Yaskawa INFORM job: A_ROOF_UPPER_0614_2_PAINT_30.JBI

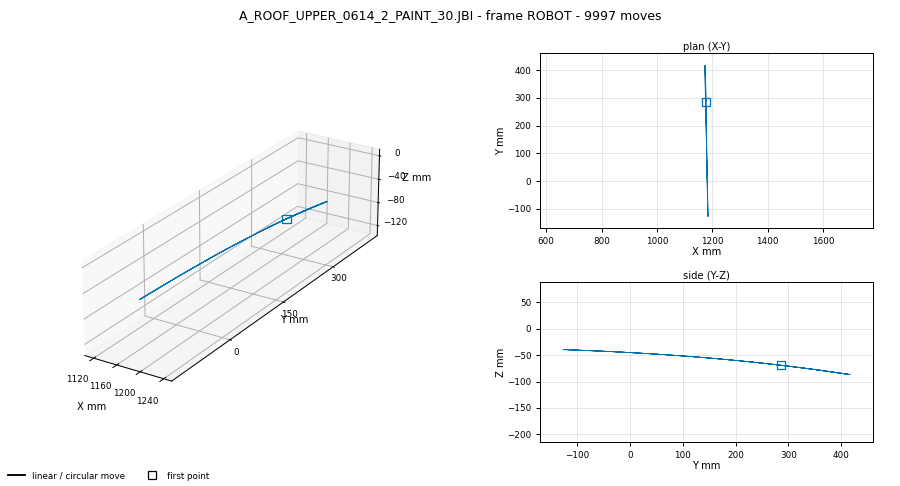
[picture p0: tool path of A_ROOF_UPPER_0614_2_PAINT_30.JBI in frame ROBOT, 9997 of 9997 moves have a stored position in this frame; points joined in program order, loops and branches not executed]
/JOB
//NAME A_ROOF_UPPER_0614_2_PAINT30
//POS
///NPOS 9997,0,0,0,0,0
///TOOL 1
///USER 0
///POSTYPE ROBOT
///RECTAN
///RCONF 1,0,0,0,0,0,0,0,0,0,0,0,0,0,0,0,0,0,0,0,0,0,0,0
C00000=1177.111,285.964,-68.993,-176.930,7.670,148.574
C00001=1177.106,286.213,-69.022,-176.928,7.672,148.574
C00002=1177.102,286.461,-69.051,-176.925,7.675,148.574
C00003=1177.098,286.710,-69.081,-176.922,7.678,148.574
C00004=1177.093,286.957,-69.110,-176.920,7.681,148.574
C00005=1177.089,287.205,-69.139,-176.917,7.684,148.574
C00006=1177.085,287.454,-69.169,-176.914,7.687,148.574
C00007=1177.081,287.702,-69.198,-176.912,7.690,148.574
C00008=1177.076,287.977,-69.230,-176.909,7.694,148.574
C00009=1177.071,288.251,-69.263,-176.906,7.697,148.574
C00010=1177.067,288.526,-69.295,-176.904,7.700,148.574
C00011=1177.062,288.801,-69.329,-176.901,7.703,148.574
C00012=1177.058,289.049,-69.358,-176.898,7.705,148.574
C00013=1177.053,289.297,-69.387,-176.896,7.708,148.574
C00014=1177.049,289.545,-69.417,-176.893,7.711,148.574
C00015=1177.045,289.793,-69.446,-176.890,7.714,148.574
C00016=1177.040,290.042,-69.476,-176.887,7.717,148.574
C00017=1177.036,290.290,-69.506,-176.885,7.720,148.574
C00018=1177.032,290.538,-69.535,-176.883,7.723,148.574
C00019=1177.027,290.787,-69.565,-176.880,7.726,148.574
C00020=1177.023,291.035,-69.594,-176.877,7.729,148.574
C00021=1177.019,291.283,-69.623,-176.875,7.732,148.574
C00022=1177.015,291.531,-69.653,-176.872,7.735,148.574
C00023=1177.011,291.780,-69.682,-176.869,7.738,148.574
C00024=1177.006,292.028,-69.713,-176.867,7.741,148.574
C00025=1177.002,292.276,-69.743,-176.865,7.743,148.574
C00026=1176.998,292.524,-69.772,-176.862,7.746,148.574
C00027=1176.994,292.772,-69.801,-176.859,7.749,148.574
C00028=1176.989,293.021,-69.831,-176.857,7.752,148.574
C00029=1176.985,293.269,-69.862,-176.854,7.755,148.574
C00030=1176.981,293.517,-69.891,-176.852,7.759,148.574
C00031=1176.976,293.765,-69.921,-176.849,7.761,148.574
C00032=1176.972,294.014,-69.950,-176.847,7.764,148.574
C00033=1176.968,294.261,-69.980,-176.844,7.767,148.574
C00034=1176.963,294.510,-70.010,-176.841,7.770,148.574
C00035=1176.959,294.758,-70.040,-176.839,7.773,148.574
C00036=1176.955,295.006,-70.070,-176.836,7.776,148.574
C00037=1176.950,295.254,-70.100,-176.834,7.779,148.574
C00038=1176.946,295.503,-70.129,-176.831,7.782,148.574
C00039=1176.942,295.750,-70.160,-176.828,7.785,148.574
C00040=1176.938,295.998,-70.189,-176.826,7.787,148.574
C00041=1176.933,296.247,-70.219,-176.824,7.790,148.574
C00042=1176.929,296.495,-70.249,-176.821,7.793,148.574
C00043=1176.925,296.743,-70.279,-176.818,7.796,148.574
C00044=1176.921,296.991,-70.309,-176.815,7.799,148.574
C00045=1176.916,297.239,-70.339,-176.813,7.802,148.574
C00046=1176.913,297.488,-70.369,-176.810,7.806,148.574
C00047=1176.908,297.736,-70.399,-176.808,7.809,148.574
C00048=1176.904,297.984,-70.429,-176.805,7.812,148.574
C00049=1176.900,298.232,-70.459,-176.803,7.814,148.574
C00050=1176.895,298.481,-70.489,-176.801,7.817,148.574
C00051=1176.891,298.728,-70.519,-176.798,7.820,148.574
C00052=1176.886,298.977,-70.549,-176.795,7.823,148.574
C00053=1176.883,299.224,-70.580,-176.792,7.826,148.574
C00054=1176.878,299.473,-70.609,-176.790,7.829,148.574
C00055=1176.874,299.721,-70.640,-176.787,7.832,148.574
C00056=1176.871,299.969,-70.670,-176.785,7.835,148.574
C00057=1176.866,300.218,-70.700,-176.782,7.838,148.574
C00058=1176.862,300.465,-70.731,-176.780,7.842,148.574
C00059=1176.857,300.714,-70.761,-176.777,7.844,148.574
C00060=1176.853,300.961,-70.791,-176.775,7.847,148.574
C00061=1176.848,301.209,-70.821,-176.772,7.850,148.574
C00062=1176.844,301.458,-70.851,-176.770,7.853,148.574
C00063=1176.840,301.706,-70.882,-176.767,7.856,148.574
C00064=1176.836,301.954,-70.912,-176.764,7.859,148.574
C00065=1176.831,302.203,-70.942,-176.762,7.862,148.574
C00066=1176.827,302.450,-70.972,-176.759,7.865,148.574
C00067=1176.823,302.698,-71.003,-176.757,7.868,148.574
C00068=1176.819,302.947,-71.033,-176.754,7.871,148.574
C00069=1176.815,303.195,-71.064,-176.751,7.874,148.574
C00070=1176.811,303.443,-71.094,-176.749,7.877,148.574
C00071=1176.806,303.691,-71.125,-176.747,7.880,148.574
C00072=1176.802,303.939,-71.155,-176.744,7.883,148.574
C00073=1176.798,304.188,-71.185,-176.742,7.886,148.575
C00074=1176.793,304.436,-71.216,-176.739,7.889,148.575
C00075=1176.789,304.683,-71.246,-176.736,7.892,148.575
C00076=1176.785,304.931,-71.277,-176.733,7.895,148.574
C00077=1176.780,305.179,-71.308,-176.731,7.898,148.575
C00078=1176.777,305.427,-71.338,-176.728,7.901,148.575
C00079=1176.772,305.676,-71.368,-176.726,7.904,148.575
C00080=1176.767,305.924,-71.399,-176.723,7.907,148.575
C00081=1176.764,306.172,-71.429,-176.721,7.910,148.575
C00082=1176.760,306.420,-71.460,-176.718,7.913,148.575
C00083=1176.755,306.668,-71.491,-176.716,7.916,148.575
C00084=1176.751,306.916,-71.521,-176.714,7.919,148.575
C00085=1176.746,307.164,-71.552,-176.711,7.922,148.575
C00086=1176.742,307.413,-71.583,-176.709,7.925,148.575
C00087=1176.739,307.660,-71.613,-176.706,7.928,148.575
C00088=1176.734,307.908,-71.644,-176.703,7.931,148.575
C00089=1176.730,308.157,-71.675,-176.701,7.935,148.575
C00090=1176.725,308.405,-71.706,-176.698,7.937,148.575
C00091=1176.721,308.652,-71.736,-176.695,7.940,148.575
C00092=1176.717,308.901,-71.767,-176.693,7.944,148.575
C00093=1176.713,309.149,-71.798,-176.690,7.947,148.575
C00094=1176.708,309.397,-71.829,-176.688,7.950,148.575
C00095=1176.704,309.645,-71.859,-176.685,7.953,148.576
C00096=1176.700,309.893,-71.890,-176.683,7.956,148.576
C00097=1176.696,310.141,-71.921,-176.680,7.959,148.576
C00098=1176.691,310.389,-71.952,-176.678,7.962,148.576
C00099=1176.688,310.637,-71.983,-176.675,7.965,148.576
C00100=1176.684,310.885,-72.014,-176.672,7.968,148.576
C00101=1176.680,311.134,-72.045,-176.671,7.971,148.576
C00102=1176.675,311.382,-72.076,-176.668,7.974,148.576
C00103=1176.670,311.629,-72.106,-176.665,7.977,148.576
C00104=1176.667,311.878,-72.138,-176.663,7.980,148.576
C00105=1176.663,312.125,-72.168,-176.660,7.983,148.576
C00106=1176.658,312.373,-72.199,-176.658,7.986,148.576
C00107=1176.654,312.622,-72.230,-176.655,7.989,148.576
C00108=1176.650,312.869,-72.262,-176.652,7.992,148.576
C00109=1176.646,313.118,-72.293,-176.650,7.996,148.576
C00110=1176.641,313.366,-72.324,-176.647,7.999,148.576
C00111=1176.637,313.613,-72.355,-176.645,8.002,148.577
C00112=1176.632,313.890,-72.389,-176.642,8.006,148.577
C00113=1176.627,314.167,-72.424,-176.639,8.009,148.577
C00114=1176.623,314.444,-72.459,-176.637,8.012,148.577
C00115=1176.618,314.721,-72.493,-176.634,8.016,148.577
C00116=1176.614,314.969,-72.525,-176.631,8.019,148.577
C00117=1176.610,315.217,-72.556,-176.629,8.022,148.577
C00118=1176.605,315.464,-72.588,-176.626,8.025,148.577
C00119=1176.601,315.713,-72.619,-176.624,8.028,148.577
C00120=1176.597,315.961,-72.649,-176.621,8.031,148.577
C00121=1176.593,316.209,-72.681,-176.619,8.035,148.577
C00122=1176.588,316.457,-72.712,-176.616,8.038,148.577
C00123=1176.585,316.705,-72.744,-176.613,8.041,148.577
C00124=1176.580,316.953,-72.775,-176.611,8.044,148.578
C00125=1176.576,317.201,-72.807,-176.608,8.047,148.577
C00126=1176.572,317.449,-72.837,-176.606,8.050,148.578
C00127=1176.568,317.697,-72.869,-176.603,8.053,148.578
C00128=1176.564,317.945,-72.900,-176.601,8.057,148.578
C00129=1176.560,318.193,-72.932,-176.598,8.060,148.578
C00130=1176.555,318.441,-72.963,-176.596,8.063,148.578
C00131=1176.551,318.689,-72.994,-176.593,8.066,148.578
C00132=1176.547,318.936,-73.026,-176.590,8.069,148.578
C00133=1176.543,319.185,-73.057,-176.588,8.072,148.578
C00134=1176.539,319.432,-73.088,-176.585,8.075,148.578
C00135=1176.535,319.681,-73.120,-176.583,8.079,148.578
C00136=1176.531,319.929,-73.151,-176.581,8.081,148.578
C00137=1176.526,320.177,-73.184,-176.579,8.084,148.579
C00138=1176.522,320.425,-73.215,-176.576,8.087,148.579
C00139=1176.518,320.673,-73.246,-176.574,8.090,148.579
C00140=1176.514,320.921,-73.278,-176.571,8.093,148.579
C00141=1176.510,321.168,-73.309,-176.569,8.097,148.579
C00142=1176.506,321.417,-73.341,-176.566,8.100,148.579
C00143=1176.501,321.664,-73.372,-176.564,8.103,148.579
C00144=1176.497,321.912,-73.404,-176.560,8.107,148.579
C00145=1176.493,322.160,-73.436,-176.558,8.110,148.579
C00146=1176.489,322.408,-73.467,-176.555,8.113,148.579
C00147=1176.485,322.656,-73.499,-176.553,8.116,148.580
C00148=1176.481,322.904,-73.530,-176.550,8.119,148.580
C00149=1176.476,323.152,-73.563,-176.548,8.123,148.580
C00150=1176.473,323.400,-73.595,-176.546,8.126,148.580
C00151=1176.468,323.648,-73.625,-176.543,8.129,148.580
C00152=1176.464,323.896,-73.657,-176.541,8.132,148.580
C00153=1176.460,324.144,-73.690,-176.538,8.135,148.580
C00154=1176.455,324.392,-73.721,-176.536,8.139,148.580
C00155=1176.452,324.640,-73.753,-176.533,8.142,148.580
C00156=1176.448,324.888,-73.785,-176.531,8.145,148.581
C00157=1176.443,325.136,-73.817,-176.528,8.148,148.581
C00158=1176.439,325.384,-73.849,-176.526,8.151,148.581
C00159=1176.436,325.632,-73.881,-176.524,8.154,148.581
C00160=1176.431,325.879,-73.913,-176.521,8.157,148.581
C00161=1176.427,326.127,-73.945,-176.519,8.161,148.581
C00162=1176.423,326.375,-73.976,-176.516,8.164,148.581
C00163=1176.418,326.623,-74.009,-176.514,8.167,148.581
C00164=1176.414,326.871,-74.040,-176.511,8.170,148.581
C00165=1176.411,327.119,-74.072,-176.509,8.173,148.582
C00166=1176.406,327.367,-74.104,-176.506,8.177,148.582
C00167=1176.402,327.615,-74.136,-176.504,8.180,148.582
C00168=1176.398,327.863,-74.168,-176.501,8.183,148.582
C00169=1176.393,328.110,-74.200,-176.499,8.186,148.582
C00170=1176.389,328.358,-74.232,-176.496,8.189,148.582
C00171=1176.385,328.607,-74.264,-176.494,8.193,148.582
C00172=1176.381,328.855,-74.296,-176.491,8.196,148.582
C00173=1176.376,329.102,-74.328,-176.489,8.199,148.583
C00174=1176.373,329.351,-74.360,-176.487,8.202,148.583
C00175=1176.369,329.598,-74.393,-176.484,8.205,148.583
C00176=1176.364,329.846,-74.425,-176.482,8.208,148.583
C00177=1176.360,330.094,-74.457,-176.480,8.212,148.583
C00178=1176.356,330.342,-74.489,-176.477,8.215,148.583
C00179=1176.352,330.590,-74.521,-176.475,8.218,148.583
C00180=1176.348,330.838,-74.554,-176.472,8.221,148.584
C00181=1176.344,331.085,-74.586,-176.470,8.224,148.584
C00182=1176.339,331.333,-74.618,-176.467,8.228,148.584
C00183=1176.336,331.581,-74.650,-176.464,8.232,148.584
C00184=1176.332,331.829,-74.683,-176.462,8.235,148.584
C00185=1176.327,332.077,-74.714,-176.459,8.238,148.584
C00186=1176.323,332.325,-74.747,-176.457,8.241,148.584
C00187=1176.319,332.572,-74.779,-176.454,8.244,148.584
C00188=1176.315,332.821,-74.812,-176.452,8.248,148.585
C00189=1176.310,333.069,-74.844,-176.450,8.251,148.585
C00190=1176.306,333.316,-74.877,-176.447,8.254,148.585
C00191=1176.302,333.564,-74.909,-176.445,8.257,148.585
C00192=1176.298,333.812,-74.941,-176.443,8.261,148.585
C00193=1176.294,334.060,-74.974,-176.440,8.264,148.585
C00194=1176.290,334.308,-75.006,-176.438,8.267,148.585
C00195=1176.286,334.556,-75.039,-176.435,8.270,148.586
C00196=1176.281,334.803,-75.071,-176.433,8.274,148.586
C00197=1176.278,335.051,-75.104,-176.430,8.277,148.586
C00198=1176.273,335.299,-75.136,-176.428,8.280,148.586
C00199=1176.269,335.547,-75.169,-176.425,8.284,148.586
C00200=1176.266,335.795,-75.201,-176.423,8.287,148.587
C00201=1176.261,336.043,-75.234,-176.420,8.290,148.587
C00202=1176.257,336.291,-75.267,-176.418,8.294,148.587
C00203=1176.254,336.538,-75.299,-176.416,8.297,148.587
C00204=1176.249,336.786,-75.331,-176.414,8.300,148.587
C00205=1176.244,337.034,-75.364,-176.411,8.303,148.587
C00206=1176.241,337.282,-75.396,-176.409,8.306,148.587
C00207=1176.237,337.529,-75.429,-176.406,8.310,148.588
C00208=1176.232,337.777,-75.463,-176.404,8.313,148.588
C00209=1176.228,338.026,-75.495,-176.402,8.316,148.588
C00210=1176.225,338.273,-75.528,-176.399,8.320,148.588
C00211=1176.220,338.521,-75.560,-176.397,8.323,148.588
C00212=1176.216,338.769,-75.593,-176.394,8.326,148.588
C00213=1176.212,339.017,-75.626,-176.392,8.330,148.589
C00214=1176.208,339.265,-75.658,-176.389,8.333,148.589
C00215=1176.204,339.513,-75.691,-176.387,8.337,148.589
C00216=1176.199,339.791,-75.729,-176.385,8.340,148.589
C00217=1176.194,340.070,-75.765,-176.381,8.344,148.589
C00218=1176.190,340.350,-75.803,-176.379,8.348,148.590
C00219=1176.185,340.628,-75.839,-176.376,8.351,148.590
C00220=1176.181,340.876,-75.872,-176.374,8.355,148.590
C00221=1176.177,341.124,-75.905,-176.372,8.358,148.590
C00222=1176.173,341.372,-75.938,-176.370,8.361,148.591
C00223=1176.168,341.620,-75.971,-176.367,8.365,148.591
C00224=1176.164,341.867,-76.004,-176.364,8.368,148.591
C00225=1176.160,342.116,-76.037,-176.362,8.372,148.591
C00226=1176.156,342.363,-76.070,-176.359,8.375,148.591
C00227=1176.152,342.611,-76.102,-176.357,8.378,148.591
C00228=1176.148,342.859,-76.136,-176.355,8.382,148.592
C00229=1176.144,343.106,-76.169,-176.353,8.385,148.592
C00230=1176.140,343.354,-76.202,-176.350,8.388,148.592
C00231=1176.136,343.602,-76.235,-176.348,8.392,148.592
C00232=1176.132,343.850,-76.268,-176.345,8.396,148.593
C00233=1176.128,344.097,-76.301,-176.343,8.399,148.593
C00234=1176.123,344.345,-76.334,-176.341,8.402,148.593
C00235=1176.119,344.593,-76.368,-176.338,8.406,148.593
C00236=1176.115,344.841,-76.400,-176.336,8.409,148.593
C00237=1176.111,345.089,-76.434,-176.334,8.412,148.594
C00238=1176.107,345.337,-76.467,-176.332,8.415,148.594
C00239=1176.103,345.584,-76.501,-176.329,8.419,148.594
C00240=1176.099,345.832,-76.534,-176.327,8.422,148.594
C00241=1176.095,346.080,-76.567,-176.324,8.426,148.595
C00242=1176.091,346.328,-76.600,-176.322,8.430,148.595
C00243=1176.087,346.575,-76.633,-176.320,8.433,148.595
C00244=1176.083,346.823,-76.666,-176.317,8.436,148.595
C00245=1176.078,347.071,-76.700,-176.315,8.439,148.595
C00246=1176.074,347.318,-76.733,-176.313,8.443,148.596
C00247=1176.070,347.566,-76.766,-176.311,8.446,148.596
C00248=1176.066,347.814,-76.799,-176.308,8.449,148.596
C00249=1176.063,348.062,-76.833,-176.305,8.453,148.596
C00250=1176.059,348.309,-76.866,-176.303,8.457,148.597
C00251=1176.054,348.557,-76.900,-176.301,8.460,148.597
C00252=1176.050,348.805,-76.933,-176.299,8.463,148.597
C00253=1176.046,349.053,-76.966,-176.296,8.467,148.597
C00254=1176.041,349.301,-77.000,-176.294,8.470,148.597
C00255=1176.038,349.548,-77.034,-176.292,8.473,148.598
C00256=1176.033,349.795,-77.067,-176.289,8.478,148.598
C00257=1176.030,350.044,-77.100,-176.287,8.481,148.598
C00258=1176.026,350.291,-77.134,-176.285,8.484,148.599
C00259=1176.021,350.539,-77.168,-176.283,8.488,148.599
C00260=1176.017,350.787,-77.201,-176.280,8.491,148.599
C00261=1176.013,351.035,-77.234,-176.278,8.494,148.599
C00262=1176.009,351.282,-77.268,-176.276,8.498,148.599
C00263=1176.006,351.530,-77.302,-176.273,8.502,148.600
C00264=1176.001,351.778,-77.335,-176.271,8.505,148.600
C00265=1175.997,352.025,-77.369,-176.269,8.509,148.600
C00266=1175.993,352.273,-77.402,-176.267,8.512,148.601
C00267=1175.989,352.520,-77.436,-176.264,8.515,148.601
C00268=1175.985,352.768,-77.470,-176.262,8.519,148.601
C00269=1175.980,353.017,-77.503,-176.260,8.522,148.601
C00270=1175.977,353.264,-77.537,-176.257,8.526,148.602
C00271=1175.972,353.511,-77.570,-176.255,8.530,148.602
C00272=1175.969,353.759,-77.605,-176.253,8.533,148.602
C00273=1175.964,354.007,-77.638,-176.251,8.537,148.603
C00274=1175.961,354.254,-77.672,-176.249,8.540,148.603
C00275=1175.956,354.502,-77.705,-176.246,8.543,148.603
C00276=1175.952,354.749,-77.740,-176.244,8.547,148.603
C00277=1175.948,354.998,-77.773,-176.242,8.551,148.604
C00278=1175.944,355.245,-77.807,-176.240,8.554,148.604
C00279=1175.941,355.492,-77.841,-176.237,8.558,148.604
C00280=1175.936,355.741,-77.875,-176.235,8.561,148.604
C00281=1175.933,355.988,-77.909,-176.233,8.565,148.605
C00282=1175.928,356.236,-77.942,-176.230,8.569,148.605
C00283=1175.924,356.483,-77.977,-176.228,8.572,148.605
C00284=1175.921,356.731,-78.011,-176.226,8.576,148.606
C00285=1175.916,356.979,-78.045,-176.224,8.579,148.606
C00286=1175.912,357.226,-78.079,-176.222,8.582,148.606
C00287=1175.908,357.475,-78.112,-176.219,8.587,148.607
C00288=1175.904,357.722,-78.147,-176.217,8.590,148.607
C00289=1175.900,357.969,-78.181,-176.215,8.593,148.607
C00290=1175.897,358.217,-78.215,-176.213,8.597,148.607
C00291=1175.892,358.465,-78.249,-176.211,8.600,148.608
C00292=1175.888,358.712,-78.282,-176.208,8.605,148.608
C00293=1175.884,358.960,-78.317,-176.206,8.608,148.608
C00294=1175.880,359.207,-78.351,-176.204,8.611,148.609
C00295=1175.875,359.455,-78.385,-176.202,8.615,148.609
C00296=1175.872,359.703,-78.419,-176.200,8.618,148.609
C00297=1175.868,359.950,-78.454,-176.198,8.622,148.610
C00298=1175.864,360.198,-78.487,-176.195,8.626,148.610
C00299=1175.860,360.446,-78.522,-176.193,8.629,148.610
C00300=1175.856,360.693,-78.555,-176.191,8.633,148.611
C00301=1175.852,360.941,-78.589,-176.189,8.636,148.611
C00302=1175.848,361.189,-78.624,-176.187,8.640,148.611
C00303=1175.844,361.436,-78.658,-176.185,8.643,148.612
C00304=1175.840,361.684,-78.693,-176.183,8.647,148.612
C00305=1175.835,361.931,-78.727,-176.181,8.651,148.613
C00306=1175.832,362.178,-78.761,-176.178,8.655,148.613
C00307=1175.828,362.427,-78.796,-176.176,8.658,148.613
C00308=1175.824,362.674,-78.830,-176.174,8.662,148.613
C00309=1175.820,362.922,-78.865,-176.172,8.665,148.614
C00310=1175.816,363.169,-78.899,-176.171,8.669,148.614
C00311=1175.812,363.417,-78.933,-176.169,8.672,148.615
C00312=1175.808,363.664,-78.967,-176.166,8.676,148.615
C00313=1175.804,363.912,-79.002,-176.164,8.680,148.615
C00314=1175.800,364.160,-79.037,-176.162,8.684,148.616
C00315=1175.796,364.407,-79.070,-176.160,8.687,148.616
C00316=1175.792,364.655,-79.105,-176.158,8.691,148.617
C00317=1175.788,364.902,-79.139,-176.156,8.694,148.617
C00318=1175.784,365.150,-79.174,-176.154,8.698,148.617
C00319=1175.779,365.398,-79.208,-176.153,8.702,148.618
C00320=1175.776,365.680,-79.248,-176.150,8.706,148.618
C00321=1175.771,365.961,-79.287,-176.148,8.710,148.619
C00322=1175.766,366.243,-79.326,-176.146,8.714,148.619
C00323=1175.761,366.525,-79.365,-176.144,8.718,148.620
C00324=1175.758,366.772,-79.400,-176.142,8.721,148.620
C00325=1175.753,367.020,-79.435,-176.140,8.725,148.621
C00326=1175.750,367.268,-79.470,-176.138,8.729,148.621
C00327=1175.746,367.515,-79.503,-176.136,8.733,148.621
C00328=1175.742,367.763,-79.538,-176.134,8.737,148.622
C00329=1175.737,368.010,-79.573,-176.134,8.740,148.622
C00330=1175.733,368.258,-79.608,-176.132,8.743,148.623
C00331=1175.730,368.505,-79.642,-176.130,8.747,148.623
C00332=1175.726,368.753,-79.677,-176.128,8.750,148.624
C00333=1175.721,369.001,-79.711,-176.126,8.754,148.624
C00334=1175.717,369.248,-79.747,-176.124,8.758,148.625
C00335=1175.714,369.496,-79.781,-176.123,8.761,148.625
C00336=1175.710,369.743,-79.816,-176.121,8.765,148.626
C00337=1175.706,369.991,-79.851,-176.119,8.769,148.626
C00338=1175.701,370.238,-79.886,-176.117,8.772,148.627
C00339=1175.697,370.486,-79.921,-176.116,8.776,148.627
C00340=1175.694,370.733,-79.955,-176.114,8.780,148.628
C00341=1175.690,370.981,-79.990,-176.112,8.784,148.628
C00342=1175.685,371.228,-80.024,-176.112,8.787,148.629
C00343=1175.682,371.476,-80.060,-176.110,8.790,148.629
C00344=1175.678,371.724,-80.095,-176.108,8.794,148.629
C00345=1175.674,371.971,-80.129,-176.107,8.798,148.630
C00346=1175.670,372.219,-80.164,-176.105,8.801,148.631
C00347=1175.666,372.466,-80.199,-176.103,8.805,148.631
C00348=1175.662,372.714,-80.234,-176.102,8.808,148.632
C00349=1175.658,372.962,-80.269,-176.101,8.812,148.632
C00350=1175.654,373.209,-80.304,-176.099,8.816,148.633
C00351=1175.650,373.457,-80.339,-176.097,8.820,148.633
C00352=1175.646,373.703,-80.374,-176.096,8.822,148.634
C00353=1175.642,373.951,-80.409,-176.095,8.826,148.634
C00354=1175.639,374.199,-80.444,-176.093,8.830,148.635
C00355=1175.634,374.446,-80.479,-176.091,8.834,148.635
C00356=1175.630,374.694,-80.514,-176.091,8.837,148.636
C00357=1175.626,374.941,-80.549,-176.089,8.841,148.637
C00358=1175.622,375.189,-80.584,-176.087,8.844,148.637
C00359=1175.618,375.437,-80.619,-176.087,8.847,148.638
C00360=1175.614,375.683,-80.654,-176.085,8.851,148.638
C00361=1175.610,375.931,-80.690,-176.084,8.854,148.639
C00362=1175.606,376.179,-80.724,-176.083,8.858,148.639
C00363=1175.602,376.426,-80.760,-176.081,8.862,148.640
C00364=1175.598,376.674,-80.795,-176.080,8.865,148.640
C00365=1175.594,376.922,-80.830,-176.079,8.869,148.641
C00366=1175.590,377.168,-80.865,-176.078,8.872,148.642
C00367=1175.586,377.416,-80.900,-176.077,8.876,148.642
C00368=1175.583,377.664,-80.936,-176.076,8.879,148.643
C00369=1175.578,377.911,-80.971,-176.074,8.883,148.643
C00370=1175.574,378.159,-81.006,-176.073,8.886,148.644
C00371=1175.571,378.406,-81.041,-176.072,8.890,148.644
C00372=1175.566,378.653,-81.076,-176.071,8.893,148.645
C00373=1175.562,378.901,-81.111,-176.070,8.897,148.646
C00374=1175.559,379.149,-81.147,-176.069,8.900,148.646
C00375=1175.555,379.396,-81.182,-176.068,8.903,148.647
C00376=1175.551,379.644,-81.217,-176.067,8.907,148.648
C00377=1175.547,379.891,-81.252,-176.066,8.910,148.648
C00378=1175.543,380.138,-81.287,-176.065,8.913,148.649
C00379=1175.539,380.386,-81.323,-176.064,8.917,148.649
C00380=1175.535,380.634,-81.358,-176.063,8.920,148.650
C00381=1175.531,380.881,-81.393,-176.062,8.923,148.651
C00382=1175.527,381.128,-81.429,-176.061,8.927,148.651
C00383=1175.523,381.375,-81.464,-176.060,8.931,148.652
C00384=1175.520,381.623,-81.500,-176.060,8.934,148.653
C00385=1175.514,381.871,-81.535,-176.059,8.937,148.653
C00386=1175.511,382.118,-81.570,-176.057,8.941,148.654
C00387=1175.507,382.366,-81.606,-176.056,8.944,148.654
C00388=1175.503,382.613,-81.641,-176.056,8.947,148.655
C00389=1175.499,382.860,-81.677,-176.055,8.950,148.656
C00390=1175.496,383.107,-81.712,-176.054,8.954,148.656
C00391=1175.492,383.356,-81.747,-176.054,8.957,148.657
C00392=1175.488,383.603,-81.782,-176.053,8.960,148.658
C00393=1175.484,383.850,-81.818,-176.052,8.963,148.658
C00394=1175.479,384.098,-81.854,-176.052,8.966,148.659
C00395=1175.476,384.345,-81.889,-176.051,8.970,148.660
C00396=1175.472,384.593,-81.925,-176.051,8.973,148.660
C00397=1175.468,384.839,-81.960,-176.050,8.976,148.661
C00398=1175.464,385.087,-81.996,-176.049,8.979,148.662
C00399=1175.460,385.335,-82.031,-176.049,8.983,148.662
C00400=1175.456,385.582,-82.067,-176.048,8.986,148.663
C00401=1175.451,385.830,-82.102,-176.047,8.989,148.664
C00402=1175.448,386.077,-82.137,-176.047,8.992,148.664
C00403=1175.444,386.325,-82.173,-176.046,8.995,148.665
C00404=1175.440,386.572,-82.208,-176.046,8.999,148.666
C00405=1175.437,386.820,-82.244,-176.045,9.001,148.666
C00406=1175.432,387.067,-82.280,-176.045,9.005,148.667
C00407=1175.428,387.314,-82.315,-176.044,9.008,148.668
C00408=1175.424,387.562,-82.351,-176.044,9.011,148.668
C00409=1175.421,387.809,-82.386,-176.044,9.014,148.669
C00410=1175.417,388.057,-82.422,-176.043,9.017,148.670
C00411=1175.412,388.304,-82.458,-176.043,9.020,148.670
C00412=1175.408,388.551,-82.493,-176.042,9.022,148.671
C00413=1175.405,388.799,-82.529,-176.042,9.026,148.672
C00414=1175.401,389.046,-82.564,-176.042,9.029,148.673
C00415=1175.397,389.294,-82.601,-176.041,9.031,148.673
C00416=1175.392,389.541,-82.636,-176.041,9.035,148.674
C00417=1175.389,389.789,-82.671,-176.041,9.037,148.675
C00418=1175.385,390.035,-82.708,-176.041,9.041,148.675
C00419=1175.382,390.283,-82.743,-176.041,9.043,148.676
C00420=1175.377,390.531,-82.779,-176.040,9.046,148.677
C00421=1175.374,390.778,-82.815,-176.040,9.049,148.677
C00422=1175.369,391.025,-82.850,-176.040,9.052,148.678
C00423=1175.366,391.273,-82.885,-176.040,9.055,148.679
C00424=1175.361,391.558,-82.927,-176.039,9.058,148.679
C00425=1175.356,391.842,-82.968,-176.039,9.062,148.680
C00426=1175.352,392.127,-83.009,-176.039,9.064,148.681
C00427=1175.348,392.411,-83.050,-176.039,9.068,148.682
C00428=1175.343,392.658,-83.086,-176.039,9.070,148.683
C00429=1175.340,392.905,-83.121,-176.039,9.074,148.683
C00430=1175.335,393.153,-83.157,-176.038,9.076,148.684
C00431=1175.332,393.401,-83.193,-176.039,9.078,148.685
C00432=1175.328,393.648,-83.228,-176.039,9.081,148.685
C00433=1175.324,393.895,-83.265,-176.038,9.084,148.686
C00434=1175.320,394.143,-83.301,-176.038,9.087,148.687
C00435=1175.316,394.390,-83.336,-176.038,9.089,148.687
C00436=1175.312,394.637,-83.372,-176.038,9.092,148.688
C00437=1175.308,394.885,-83.408,-176.039,9.094,148.689
C00438=1175.304,395.133,-83.443,-176.038,9.098,148.690
C00439=1175.301,395.379,-83.479,-176.038,9.100,148.690
C00440=1175.296,395.627,-83.516,-176.038,9.103,148.691
C00441=1175.293,395.875,-83.551,-176.038,9.105,148.692
C00442=1175.288,396.122,-83.586,-176.038,9.108,148.692
C00443=1175.284,396.369,-83.623,-176.039,9.110,148.693
C00444=1175.281,396.616,-83.659,-176.038,9.113,148.693
C00445=1175.277,396.864,-83.694,-176.038,9.115,148.694
C00446=1175.273,397.112,-83.730,-176.039,9.118,148.695
C00447=1175.269,397.359,-83.766,-176.039,9.120,148.696
C00448=1175.265,397.607,-83.802,-176.039,9.123,148.696
C00449=1175.261,397.853,-83.838,-176.039,9.125,148.697
C00450=1175.257,398.100,-83.874,-176.039,9.128,148.698
C00451=1175.253,398.348,-83.910,-176.039,9.130,148.698
C00452=1175.249,398.596,-83.945,-176.039,9.133,148.699
C00453=1175.245,398.843,-83.981,-176.039,9.135,148.700
C00454=1175.241,399.091,-84.018,-176.039,9.138,148.700
C00455=1175.238,399.338,-84.053,-176.039,9.140,148.701
C00456=1175.234,399.586,-84.089,-176.039,9.143,148.702
C00457=1175.229,399.833,-84.125,-176.040,9.144,148.702
C00458=1175.225,400.079,-84.161,-176.040,9.147,148.703
C00459=1175.222,400.327,-84.196,-176.040,9.149,148.704
C00460=1175.217,400.575,-84.233,-176.040,9.152,148.704
C00461=1175.214,400.822,-84.269,-176.040,9.154,148.705
C00462=1175.210,401.069,-84.305,-176.040,9.157,148.706
C00463=1175.206,401.317,-84.340,-176.041,9.159,148.706
C00464=1175.202,401.564,-84.376,-176.041,9.161,148.707
C00465=1175.198,401.812,-84.413,-176.041,9.163,148.707
C00466=1175.195,402.059,-84.448,-176.041,9.166,148.708
C00467=1175.190,402.306,-84.484,-176.042,9.168,148.709
C00468=1175.186,402.554,-84.520,-176.041,9.170,148.709
C00469=1175.183,402.801,-84.556,-176.041,9.172,148.710
C00470=1175.178,403.048,-84.592,-176.042,9.175,148.711
C00471=1175.175,403.296,-84.628,-176.042,9.176,148.711
C00472=1175.171,403.543,-84.664,-176.042,9.179,148.712
C00473=1175.167,403.791,-84.700,-176.042,9.182,148.713
C00474=1175.163,404.038,-84.736,-176.042,9.183,148.713
C00475=1175.159,404.285,-84.773,-176.043,9.186,148.714
C00476=1175.155,404.533,-84.808,-176.043,9.188,148.715
C00477=1175.151,404.781,-84.844,-176.043,9.190,148.715
C00478=1175.147,405.027,-84.880,-176.043,9.192,148.716
C00479=1175.143,405.274,-84.916,-176.043,9.194,148.716
C00480=1175.139,405.522,-84.952,-176.044,9.196,148.717
C00481=1175.136,405.769,-84.988,-176.044,9.199,148.718
C00482=1175.131,406.017,-85.024,-176.044,9.200,148.718
C00483=1175.127,406.264,-85.060,-176.044,9.203,148.719
C00484=1175.124,406.511,-85.096,-176.044,9.205,148.719
C00485=1175.120,406.759,-85.132,-176.045,9.207,148.720
C00486=1175.116,407.007,-85.168,-176.045,9.209,148.721
C00487=1175.112,407.254,-85.205,-176.045,9.211,148.721
C00488=1175.108,407.501,-85.240,-176.045,9.213,148.722
C00489=1175.104,407.749,-85.276,-176.046,9.215,148.722
C00490=1175.101,407.996,-85.313,-176.046,9.217,148.723
C00491=1175.096,408.243,-85.348,-176.046,9.219,148.723
C00492=1175.092,408.490,-85.385,-176.046,9.221,148.724
C00493=1175.089,408.737,-85.420,-176.047,9.223,148.725
C00494=1175.084,408.985,-85.456,-176.047,9.225,148.725
C00495=1175.081,409.232,-85.493,-176.047,9.227,148.726
C00496=1175.076,409.480,-85.529,-176.047,9.229,148.726
C00497=1175.073,409.727,-85.564,-176.047,9.231,148.727
C00498=1175.069,409.975,-85.601,-176.048,9.233,148.728
C00499=1175.065,410.222,-85.637,-176.048,9.235,148.728
C00500=1175.062,410.469,-85.673,-176.048,9.237,148.729
C00501=1175.057,410.717,-85.709,-176.048,9.239,148.729
C00502=1175.054,410.964,-85.745,-176.048,9.241,148.730
C00503=1175.049,411.211,-85.781,-176.049,9.243,148.730
C00504=1175.046,411.459,-85.817,-176.048,9.245,148.731
C00505=1175.042,411.706,-85.854,-176.049,9.247,148.732
C00506=1175.038,411.954,-85.889,-176.049,9.248,148.732
C00507=1175.033,412.201,-85.925,-176.049,9.251,148.733
C00508=1175.030,412.448,-85.961,-176.050,9.252,148.733
C00509=1175.025,412.695,-85.998,-176.050,9.255,148.734
C00510=1175.022,412.942,-86.034,-176.050,9.256,148.734
C00511=1175.018,413.190,-86.070,-176.050,9.259,148.735
C00512=1175.014,413.437,-86.106,-176.050,9.260,148.735
C00513=1175.010,413.685,-86.142,-176.051,9.261,148.736
C00514=1175.006,413.932,-86.178,-176.051,9.264,148.737
C00515=1175.002,414.180,-86.215,-176.051,9.265,148.737
C00516=1174.998,414.427,-86.250,-176.051,9.268,148.738
C00517=1174.995,414.674,-86.287,-176.052,9.269,148.738
C00518=1174.991,414.922,-86.323,-176.052,9.271,148.739
C00519=1174.987,415.169,-86.359,-176.052,9.273,148.739
C00520=1174.983,415.416,-86.395,-176.052,9.275,148.740
C00521=1174.979,415.663,-86.431,-176.053,9.276,148.740
C00522=1174.976,415.912,-86.467,-176.052,9.279,148.741
C00523=1174.975,416.158,-86.503,-176.053,9.280,148.741
C00524=1174.975,416.409,-86.539,-176.053,9.281,148.742
C00525=1174.975,416.659,-86.575,-176.053,9.284,148.742
C00526=1174.978,416.908,-86.611,-176.053,9.285,148.743
C00527=1174.981,417.157,-86.647,-176.053,9.287,148.743
C00528=1174.559,417.159,-86.691,-176.056,9.298,148.747
C00529=1174.556,416.906,-86.655,-176.056,9.296,148.746
C00530=1174.555,416.654,-86.619,-176.056,9.295,148.746
C00531=1174.554,416.401,-86.582,-176.056,9.292,148.745
C00532=1174.554,416.147,-86.545,-176.056,9.291,148.745
C00533=1174.556,415.900,-86.509,-176.055,9.289,148.744
C00534=1174.558,415.652,-86.473,-176.055,9.287,148.744
C00535=1174.562,415.405,-86.438,-176.055,9.286,148.743
C00536=1174.566,415.158,-86.401,-176.055,9.284,148.743
C00537=1174.569,414.910,-86.365,-176.055,9.282,148.742
C00538=1174.573,414.663,-86.328,-176.054,9.280,148.742
C00539=1174.577,414.416,-86.293,-176.054,9.279,148.741
C00540=1174.581,414.168,-86.256,-176.054,9.276,148.741
C00541=1174.585,413.921,-86.220,-176.054,9.275,148.740
C00542=1174.589,413.674,-86.184,-176.054,9.272,148.740
C00543=1174.593,413.426,-86.148,-176.054,9.271,148.739
C00544=1174.597,413.178,-86.112,-176.053,9.269,148.739
C00545=1174.600,412.931,-86.076,-176.053,9.267,148.738
C00546=1174.605,412.684,-86.039,-176.053,9.265,148.737
C00547=1174.608,412.437,-86.003,-176.053,9.263,148.737
C00548=1174.613,412.189,-85.967,-176.053,9.262,148.736
C00549=1174.616,411.943,-85.931,-176.052,9.260,148.736
C00550=1174.621,411.695,-85.895,-176.052,9.258,148.735
C00551=1174.625,411.447,-85.859,-176.052,9.256,148.735
C00552=1174.629,411.200,-85.823,-176.052,9.254,148.734
C00553=1174.632,410.953,-85.787,-176.051,9.252,148.734
C00554=1174.636,410.706,-85.750,-176.051,9.250,148.733
C00555=1174.640,410.458,-85.715,-176.051,9.248,148.732
C00556=1174.643,410.211,-85.678,-176.051,9.246,148.732
C00557=1174.648,409.963,-85.642,-176.050,9.244,148.731
C00558=1174.651,409.716,-85.607,-176.050,9.242,148.731
C00559=1174.656,409.469,-85.570,-176.050,9.240,148.730
C00560=1174.659,409.221,-85.534,-176.049,9.238,148.729
C00561=1174.663,408.974,-85.497,-176.050,9.236,148.729
C00562=1174.667,408.727,-85.462,-176.049,9.234,148.728
C00563=1174.671,408.479,-85.426,-176.049,9.232,148.728
C00564=1174.675,408.232,-85.389,-176.048,9.230,148.727
C00565=1174.678,407.984,-85.354,-176.049,9.228,148.727
C00566=1174.683,407.737,-85.318,-176.048,9.226,148.726
C00567=1174.687,407.490,-85.282,-176.048,9.224,148.725
C00568=1174.691,407.243,-85.246,-176.048,9.222,148.725
C00569=1174.695,406.996,-85.209,-176.048,9.220,148.724
C00570=1174.699,406.748,-85.173,-176.048,9.217,148.724
C00571=1174.703,406.500,-85.138,-176.047,9.216,148.723
C00572=1174.707,406.253,-85.101,-176.047,9.213,148.722
C00573=1174.710,406.006,-85.065,-176.046,9.212,148.722
C00574=1174.714,405.758,-85.030,-176.047,9.209,148.721
C00575=1174.718,405.511,-84.993,-176.046,9.208,148.721
C00576=1174.722,405.263,-84.957,-176.046,9.205,148.720
C00577=1174.726,405.016,-84.921,-176.046,9.203,148.719
C00578=1174.730,404.769,-84.885,-176.045,9.201,148.719
C00579=1174.734,404.522,-84.850,-176.046,9.199,148.718
C00580=1174.738,404.274,-84.814,-176.046,9.196,148.717
C00581=1174.742,404.027,-84.777,-176.045,9.195,148.717
C00582=1174.746,403.779,-84.741,-176.045,9.192,148.716
C00583=1174.750,403.532,-84.706,-176.045,9.190,148.716
C00584=1174.754,403.285,-84.669,-176.044,9.188,148.715
C00585=1174.757,403.037,-84.633,-176.044,9.186,148.714
C00586=1174.761,402.790,-84.598,-176.044,9.183,148.714
C00587=1174.765,402.543,-84.561,-176.044,9.181,148.713
C00588=1174.769,402.295,-84.525,-176.043,9.179,148.712
C00589=1174.773,402.047,-84.489,-176.044,9.177,148.712
C00590=1174.777,401.801,-84.453,-176.043,9.175,148.711
C00591=1174.781,401.554,-84.418,-176.043,9.172,148.710
C00592=1174.785,401.306,-84.382,-176.043,9.170,148.710
C00593=1174.789,401.058,-84.346,-176.043,9.167,148.709
C00594=1174.793,400.811,-84.309,-176.043,9.165,148.708
C00595=1174.797,400.564,-84.274,-176.042,9.163,148.708
C00596=1174.800,400.316,-84.238,-176.042,9.161,148.707
C00597=1174.804,400.069,-84.201,-176.042,9.158,148.707
C00598=1174.808,399.821,-84.166,-176.042,9.156,148.706
C00599=1174.812,399.574,-84.130,-176.042,9.153,148.705
C00600=1174.817,399.327,-84.094,-176.042,9.151,148.705
C00601=1174.820,399.080,-84.058,-176.041,9.149,148.704
C00602=1174.824,398.832,-84.022,-176.041,9.147,148.703
C00603=1174.828,398.585,-83.986,-176.041,9.144,148.702
C00604=1174.832,398.337,-83.951,-176.041,9.141,148.702
C00605=1174.836,398.090,-83.914,-176.041,9.139,148.701
C00606=1174.840,397.842,-83.878,-176.041,9.137,148.701
C00607=1174.843,397.595,-83.843,-176.041,9.134,148.700
C00608=1174.848,397.348,-83.807,-176.041,9.132,148.699
C00609=1174.852,397.100,-83.772,-176.041,9.129,148.698
C00610=1174.855,396.853,-83.735,-176.041,9.127,148.698
C00611=1174.860,396.606,-83.699,-176.041,9.124,148.697
C00612=1174.863,396.358,-83.664,-176.041,9.122,148.696
C00613=1174.867,396.111,-83.628,-176.040,9.119,148.696
C00614=1174.871,395.863,-83.591,-176.040,9.116,148.695
C00615=1174.875,395.616,-83.556,-176.040,9.114,148.694
C00616=1174.879,395.369,-83.521,-176.040,9.112,148.694
C00617=1174.883,395.121,-83.484,-176.041,9.108,148.693
C00618=1174.887,394.874,-83.449,-176.041,9.106,148.692
C00619=1174.891,394.626,-83.413,-176.040,9.103,148.692
C00620=1174.895,394.379,-83.376,-176.041,9.101,148.691
C00621=1174.898,394.132,-83.341,-176.041,9.098,148.690
C00622=1174.902,393.884,-83.305,-176.040,9.096,148.690
C00623=1174.907,393.637,-83.270,-176.041,9.092,148.689
C00624=1174.911,393.390,-83.234,-176.041,9.090,148.688
C00625=1174.914,393.142,-83.198,-176.040,9.087,148.687
C00626=1174.919,392.895,-83.162,-176.041,9.085,148.687
C00627=1174.922,392.647,-83.126,-176.041,9.081,148.686
C00628=1174.926,392.400,-83.090,-176.041,9.079,148.685
C00629=1174.931,392.115,-83.049,-176.041,9.075,148.685
C00630=1174.935,391.831,-83.009,-176.041,9.073,148.684
C00631=1174.940,391.546,-82.968,-176.041,9.069,148.683
C00632=1174.945,391.262,-82.926,-176.042,9.066,148.682
C00633=1174.948,391.014,-82.890,-176.042,9.064,148.682
C00634=1174.952,390.767,-82.855,-176.042,9.060,148.681
C00635=1174.956,390.519,-82.819,-176.042,9.058,148.680
C00636=1174.960,390.272,-82.783,-176.042,9.054,148.679
C00637=1174.964,390.025,-82.748,-176.043,9.052,148.679
C00638=1174.968,389.777,-82.712,-176.043,9.049,148.678
C00639=1174.972,389.530,-82.677,-176.043,9.046,148.677
C00640=1174.976,389.282,-82.641,-176.043,9.043,148.677
C00641=1174.980,389.035,-82.605,-176.044,9.040,148.676
C00642=1174.983,388.787,-82.570,-176.044,9.037,148.675
C00643=1174.987,388.541,-82.534,-176.044,9.034,148.674
C00644=1174.992,388.293,-82.498,-176.045,9.031,148.674
C00645=1174.995,388.046,-82.462,-176.045,9.028,148.673
C00646=1174.999,387.798,-82.426,-176.046,9.024,148.672
C00647=1175.003,387.551,-82.391,-176.046,9.022,148.672
C00648=1175.007,387.304,-82.356,-176.046,9.019,148.671
C00649=1175.011,387.056,-82.320,-176.047,9.015,148.670
C00650=1175.015,386.808,-82.284,-176.047,9.012,148.670
C00651=1175.019,386.561,-82.249,-176.047,9.010,148.669
C00652=1175.022,386.313,-82.213,-176.048,9.007,148.668
C00653=1175.027,386.067,-82.178,-176.049,9.003,148.668
C00654=1175.031,385.819,-82.142,-176.049,9.000,148.667
C00655=1175.035,385.571,-82.107,-176.050,8.997,148.666
C00656=1175.039,385.323,-82.071,-176.051,8.994,148.666
C00657=1175.043,385.076,-82.036,-176.051,8.990,148.665
C00658=1175.047,384.829,-82.001,-176.052,8.987,148.664
C00659=1175.050,384.581,-81.965,-176.052,8.984,148.664
C00660=1175.055,384.334,-81.929,-176.053,8.981,148.663
C00661=1175.058,384.086,-81.893,-176.053,8.977,148.662
C00662=1175.062,383.839,-81.858,-176.054,8.974,148.662
C00663=1175.066,383.592,-81.823,-176.055,8.971,148.661
C00664=1175.070,383.344,-81.787,-176.056,8.968,148.660
C00665=1175.073,383.097,-81.751,-176.056,8.965,148.660
C00666=1175.078,382.849,-81.717,-176.057,8.961,148.659
C00667=1175.082,382.602,-81.681,-176.058,8.958,148.658
C00668=1175.086,382.354,-81.645,-176.058,8.955,148.658
C00669=1175.090,382.107,-81.610,-176.060,8.951,148.657
C00670=1175.094,381.860,-81.575,-176.060,8.948,148.656
C00671=1175.098,381.612,-81.539,-176.061,8.945,148.656
C00672=1175.102,381.364,-81.504,-176.062,8.942,148.655
C00673=1175.106,381.117,-81.469,-176.063,8.939,148.655
C00674=1175.110,380.870,-81.433,-176.064,8.934,148.654
C00675=1175.113,380.622,-81.398,-176.065,8.931,148.653
C00676=1175.117,380.375,-81.362,-176.065,8.928,148.653
C00677=1175.121,380.127,-81.328,-176.067,8.924,148.652
C00678=1175.126,379.880,-81.292,-176.068,8.921,148.652
C00679=1175.130,379.632,-81.256,-176.068,8.918,148.651
C00680=1175.134,379.385,-81.221,-176.070,8.914,148.650
C00681=1175.138,379.137,-81.186,-176.071,8.911,148.650
C00682=1175.141,378.890,-81.151,-176.072,8.907,148.649
C00683=1175.146,378.643,-81.115,-176.073,8.904,148.649
C00684=1175.149,378.395,-81.080,-176.074,8.901,148.648
C00685=1175.153,378.147,-81.045,-176.075,8.897,148.647
C00686=1175.157,377.900,-81.010,-176.076,8.894,148.647
C00687=1175.161,377.653,-80.974,-176.077,8.890,148.646
C00688=1175.165,377.405,-80.940,-176.078,8.887,148.646
C00689=1175.169,377.157,-80.904,-176.080,8.883,148.645
C00690=1175.173,376.911,-80.869,-176.081,8.879,148.644
C00691=1175.177,376.662,-80.834,-176.082,8.876,148.644
C00692=1175.181,376.415,-80.798,-176.083,8.872,148.643
C00693=1175.185,376.168,-80.764,-176.085,8.869,148.643
C00694=1175.189,375.920,-80.728,-176.086,8.865,148.642
C00695=1175.193,375.673,-80.693,-176.087,8.862,148.641
C00696=1175.197,375.425,-80.658,-176.088,8.858,148.641
C00697=1175.201,375.178,-80.623,-176.090,8.854,148.640
C00698=1175.205,374.930,-80.588,-176.091,8.852,148.640
C00699=1175.208,374.683,-80.553,-176.092,8.848,148.639
C00700=1175.212,374.435,-80.519,-176.094,8.844,148.639
C00701=1175.217,374.188,-80.483,-176.096,8.840,148.638
C00702=1175.221,373.940,-80.449,-176.096,8.837,148.638
C00703=1175.224,373.692,-80.413,-176.098,8.834,148.637
C00704=1175.229,373.445,-80.379,-176.100,8.830,148.636
C00705=1175.233,373.198,-80.343,-176.100,8.827,148.636
C00706=1175.237,372.950,-80.309,-176.102,8.823,148.635
C00707=1175.241,372.703,-80.273,-176.104,8.819,148.635
C00708=1175.245,372.454,-80.238,-176.105,8.815,148.634
C00709=1175.248,372.208,-80.204,-176.107,8.811,148.634
C00710=1175.252,371.960,-80.169,-176.108,8.809,148.633
C00711=1175.256,371.713,-80.134,-176.110,8.805,148.633
C00712=1175.260,371.465,-80.099,-176.111,8.801,148.632
C00713=1175.264,371.217,-80.064,-176.113,8.798,148.632
C00714=1175.269,370.970,-80.029,-176.115,8.794,148.631
C00715=1175.272,370.722,-79.994,-176.116,8.790,148.631
C00716=1175.276,370.475,-79.959,-176.118,8.786,148.630
C00717=1175.280,370.227,-79.924,-176.120,8.783,148.630
C00718=1175.285,369.980,-79.890,-176.121,8.780,148.629
C00719=1175.288,369.732,-79.854,-176.123,8.776,148.629
C00720=1175.292,369.485,-79.821,-176.125,8.772,148.629
C00721=1175.296,369.237,-79.786,-176.126,8.769,148.628
C00722=1175.301,368.990,-79.751,-176.128,8.765,148.627
C00723=1175.304,368.742,-79.716,-176.130,8.761,148.627
C00724=1175.308,368.494,-79.682,-176.132,8.758,148.627
C00725=1175.312,368.247,-79.647,-176.133,8.754,148.626
C00726=1175.316,368.000,-79.611,-176.135,8.751,148.626
C00727=1175.320,367.752,-79.577,-176.137,8.747,148.625
C00728=1175.324,367.504,-79.543,-176.138,8.743,148.625
C00729=1175.328,367.257,-79.508,-176.140,8.739,148.624
C00730=1175.332,367.009,-79.473,-176.142,8.736,148.624
C00731=1175.336,366.762,-79.438,-176.144,8.732,148.623
C00732=1175.340,366.514,-79.404,-176.146,8.729,148.623
C00733=1175.345,366.233,-79.365,-176.148,8.724,148.622
C00734=1175.350,365.950,-79.326,-176.150,8.720,148.622
C00735=1175.354,365.668,-79.286,-176.152,8.716,148.622
C00736=1175.358,365.387,-79.247,-176.155,8.712,148.621
C00737=1175.363,365.139,-79.213,-176.157,8.708,148.621
C00738=1175.367,364.891,-79.178,-176.159,8.705,148.620
C00739=1175.371,364.644,-79.144,-176.161,8.701,148.620
C00740=1175.374,364.396,-79.108,-176.163,8.697,148.620
C00741=1175.378,364.149,-79.075,-176.164,8.694,148.619
C00742=1175.382,363.901,-79.040,-176.166,8.690,148.619
C00743=1175.387,363.654,-79.005,-176.169,8.687,148.619
C00744=1175.390,363.406,-78.971,-176.171,8.682,148.618
C00745=1175.394,363.159,-78.937,-176.173,8.679,148.618
C00746=1175.398,362.911,-78.903,-176.175,8.675,148.617
C00747=1175.402,362.663,-78.868,-176.177,8.672,148.617
C00748=1175.406,362.416,-78.834,-176.179,8.668,148.617
C00749=1175.410,362.168,-78.799,-176.181,8.665,148.616
C00750=1175.415,361.920,-78.765,-176.183,8.661,148.616
C00751=1175.418,361.672,-78.731,-176.185,8.657,148.615
C00752=1175.423,361.425,-78.697,-176.188,8.654,148.615
C00753=1175.427,361.178,-78.663,-176.189,8.650,148.615
C00754=1175.430,360.930,-78.628,-176.191,8.646,148.614
C00755=1175.434,360.682,-78.594,-176.193,8.643,148.614
C00756=1175.439,360.435,-78.560,-176.195,8.640,148.614
C00757=1175.442,360.187,-78.525,-176.198,8.636,148.613
C00758=1175.447,359.939,-78.492,-176.200,8.632,148.613
C00759=1175.450,359.691,-78.457,-176.202,8.628,148.613
C00760=1175.454,359.444,-78.424,-176.204,8.625,148.612
C00761=1175.459,359.197,-78.389,-176.206,8.622,148.612
C00762=1175.462,358.949,-78.355,-176.209,8.618,148.612
C00763=1175.467,358.701,-78.321,-176.211,8.614,148.611
C00764=1175.471,358.454,-78.287,-176.213,8.611,148.611
C00765=1175.475,358.206,-78.252,-176.215,8.607,148.611
C00766=1175.478,357.959,-78.219,-176.217,8.604,148.611
C00767=1175.482,357.711,-78.185,-176.219,8.600,148.610
C00768=1175.486,357.463,-78.151,-176.222,8.596,148.610
C00769=1175.490,357.216,-78.117,-176.224,8.593,148.610
C00770=1175.495,356.968,-78.083,-176.226,8.589,148.609
C00771=1175.498,356.720,-78.049,-176.228,8.586,148.609
C00772=1175.502,356.473,-78.015,-176.231,8.582,148.609
C00773=1175.507,356.225,-77.981,-176.233,8.579,148.608
C00774=1175.511,355.978,-77.947,-176.235,8.575,148.608
C00775=1175.514,355.729,-77.914,-176.238,8.571,148.608
C00776=1175.519,355.482,-77.879,-176.240,8.568,148.608
C00777=1175.523,355.235,-77.845,-176.242,8.564,148.607
C00778=1175.526,354.986,-77.812,-176.244,8.561,148.607
C00779=1175.531,354.739,-77.777,-176.247,8.557,148.607
C00780=1175.535,354.491,-77.744,-176.249,8.553,148.606
C00781=1175.539,354.244,-77.710,-176.251,8.550,148.606
C00782=1175.543,353.995,-77.676,-176.253,8.547,148.606
C00783=1175.547,353.748,-77.642,-176.256,8.543,148.606
C00784=1175.551,353.500,-77.609,-176.257,8.540,148.605
C00785=1175.555,353.253,-77.575,-176.260,8.536,148.605
C00786=1175.559,353.005,-77.541,-176.262,8.532,148.605
C00787=1175.563,352.757,-77.507,-176.265,8.529,148.604
C00788=1175.567,352.510,-77.474,-176.267,8.526,148.604
C00789=1175.571,352.262,-77.441,-176.269,8.522,148.604
C00790=1175.576,352.015,-77.407,-176.271,8.519,148.604
C00791=1175.580,351.766,-77.373,-176.274,8.515,148.603
C00792=1175.583,351.519,-77.339,-176.276,8.511,148.603
C00793=1175.587,351.271,-77.306,-176.279,8.508,148.603
C00794=1175.592,351.024,-77.273,-176.281,8.505,148.603
C00795=1175.596,350.776,-77.238,-176.283,8.501,148.602
C00796=1175.600,350.528,-77.205,-176.285,8.498,148.602
C00797=1175.604,350.280,-77.172,-176.288,8.494,148.602
C00798=1175.608,350.033,-77.138,-176.290,8.490,148.602
C00799=1175.612,349.785,-77.105,-176.292,8.487,148.601
C00800=1175.616,349.537,-77.072,-176.295,8.484,148.601
C00801=1175.621,349.289,-77.038,-176.297,8.480,148.601
C00802=1175.625,349.042,-77.004,-176.299,8.477,148.601
C00803=1175.628,348.794,-76.970,-176.301,8.474,148.600
C00804=1175.632,348.546,-76.937,-176.304,8.469,148.600
C00805=1175.637,348.298,-76.904,-176.306,8.466,148.600
C00806=1175.641,348.051,-76.871,-176.308,8.463,148.600
C00807=1175.644,347.804,-76.837,-176.311,8.460,148.599
C00808=1175.649,347.556,-76.804,-176.313,8.456,148.599
C00809=1175.653,347.308,-76.771,-176.315,8.453,148.599
C00810=1175.657,347.060,-76.738,-176.317,8.450,148.599
C00811=1175.661,346.813,-76.704,-176.320,8.445,148.598
C00812=1175.665,346.564,-76.671,-176.323,8.442,148.598
C00813=1175.669,346.316,-76.638,-176.325,8.439,148.598
C00814=1175.674,346.068,-76.604,-176.327,8.436,148.598
C00815=1175.678,345.821,-76.571,-176.329,8.432,148.598
C00816=1175.682,345.573,-76.538,-176.332,8.429,148.597
C00817=1175.686,345.325,-76.505,-176.334,8.426,148.597
C00818=1175.690,345.078,-76.471,-176.336,8.422,148.597
C00819=1175.694,344.830,-76.438,-176.339,8.418,148.597
C00820=1175.698,344.583,-76.404,-176.341,8.415,148.596
C00821=1175.702,344.335,-76.373,-176.344,8.412,148.596
C00822=1175.706,344.087,-76.339,-176.346,8.408,148.596
C00823=1175.710,343.839,-76.306,-176.348,8.405,148.596
C00824=1175.714,343.591,-76.273,-176.350,8.402,148.596
C00825=1175.718,343.344,-76.240,-176.353,8.398,148.595
C00826=1175.722,343.096,-76.207,-176.355,8.395,148.595
C00827=1175.727,342.848,-76.174,-176.358,8.391,148.595
C00828=1175.731,342.601,-76.140,-176.361,8.388,148.595
C00829=1175.735,342.353,-76.107,-176.363,8.385,148.595
C00830=1175.739,342.105,-76.074,-176.365,8.381,148.594
C00831=1175.743,341.857,-76.041,-176.367,8.378,148.594
C00832=1175.748,341.609,-76.009,-176.370,8.375,148.594
C00833=1175.752,341.361,-75.975,-176.372,8.371,148.594
C00834=1175.755,341.114,-75.943,-176.374,8.368,148.594
C00835=1175.759,340.866,-75.910,-176.376,8.365,148.593
C00836=1175.763,340.618,-75.876,-176.379,8.361,148.593
C00837=1175.768,340.338,-75.840,-176.382,8.358,148.593
C00838=1175.773,340.060,-75.803,-176.385,8.354,148.593
C00839=1175.777,339.780,-75.766,-176.387,8.350,148.593
C00840=1175.782,339.501,-75.729,-176.390,8.346,148.592
C00841=1175.786,339.254,-75.696,-176.392,8.343,148.592
C00842=1175.790,339.005,-75.663,-176.394,8.339,148.592
C00843=1175.795,338.758,-75.630,-176.397,8.336,148.592
C00844=1175.799,338.510,-75.597,-176.399,8.333,148.592
C00845=1175.802,338.262,-75.565,-176.402,8.330,148.592
C00846=1175.807,338.014,-75.532,-176.404,8.327,148.591
C00847=1175.811,337.766,-75.499,-176.407,8.322,148.591
C00848=1175.815,337.518,-75.467,-176.410,8.319,148.591
C00849=1175.819,337.271,-75.434,-176.412,8.316,148.591
C00850=1175.824,337.023,-75.402,-176.414,8.313,148.591
C00851=1175.828,336.775,-75.369,-176.416,8.310,148.590
C00852=1175.831,336.528,-75.336,-176.419,8.306,148.590
C00853=1175.836,336.280,-75.304,-176.421,8.303,148.590
C00854=1175.840,336.032,-75.271,-176.424,8.300,148.590
C00855=1175.843,335.784,-75.239,-176.426,8.297,148.590
C00856=1175.848,335.536,-75.206,-176.428,8.293,148.590
C00857=1175.852,335.288,-75.173,-176.431,8.290,148.590
C00858=1175.856,335.041,-75.141,-176.433,8.287,148.589
C00859=1175.860,334.793,-75.108,-176.435,8.284,148.589
C00860=1175.865,334.545,-75.075,-176.438,8.280,148.589
C00861=1175.868,334.297,-75.043,-176.441,8.277,148.589
C00862=1175.872,334.049,-75.010,-176.443,8.273,148.589
C00863=1175.876,333.801,-74.978,-176.446,8.270,148.589
C00864=1175.881,333.553,-74.946,-176.448,8.267,148.588
C00865=1175.885,333.306,-74.913,-176.451,8.264,148.588
C00866=1175.889,333.058,-74.881,-176.453,8.260,148.588
C00867=1175.893,332.809,-74.849,-176.455,8.257,148.588
C00868=1175.897,332.562,-74.816,-176.458,8.254,148.588
C00869=1175.901,332.314,-74.784,-176.460,8.251,148.588
C00870=1175.906,332.066,-74.752,-176.462,8.247,148.587
C00871=1175.910,331.818,-74.719,-176.465,8.244,148.587
C00872=1175.913,331.570,-74.687,-176.467,8.241,148.587
C00873=1175.918,331.322,-74.655,-176.470,8.238,148.587
C00874=1175.923,331.075,-74.622,-176.472,8.235,148.587
C00875=1175.926,330.827,-74.590,-176.475,8.232,148.587
C00876=1175.931,330.579,-74.558,-176.477,8.227,148.587
C00877=1175.935,330.331,-74.526,-176.480,8.224,148.587
C00878=1175.939,330.083,-74.495,-176.482,8.221,148.586
C00879=1175.943,329.836,-74.461,-176.485,8.218,148.586
C00880=1175.947,329.588,-74.430,-176.487,8.215,148.586
C00881=1175.951,329.339,-74.397,-176.490,8.211,148.586
C00882=1175.955,329.092,-74.366,-176.492,8.208,148.586
C00883=1175.960,328.843,-74.333,-176.495,8.205,148.586
C00884=1175.964,328.595,-74.301,-176.497,8.202,148.586
C00885=1175.968,328.348,-74.268,-176.499,8.199,148.585
C00886=1175.972,328.100,-74.237,-176.502,8.196,148.585
C00887=1175.976,327.852,-74.205,-176.504,8.192,148.585
C00888=1175.980,327.604,-74.173,-176.507,8.189,148.585
C00889=1175.984,327.357,-74.141,-176.509,8.186,148.585
C00890=1175.989,327.108,-74.109,-176.512,8.183,148.585
C00891=1175.993,326.860,-74.077,-176.514,8.180,148.585
C00892=1175.996,326.612,-74.045,-176.517,8.176,148.585
C00893=1176.001,326.365,-74.013,-176.519,8.173,148.585
C00894=1176.005,326.117,-73.981,-176.522,8.170,148.584
C00895=1176.009,325.868,-73.949,-176.524,8.167,148.584
C00896=1176.014,325.621,-73.917,-176.527,8.164,148.584
C00897=1176.018,325.373,-73.885,-176.529,8.160,148.584
C00898=1176.021,325.125,-73.853,-176.532,8.157,148.584
C00899=1176.026,324.877,-73.821,-176.534,8.154,148.584
C00900=1176.030,324.629,-73.789,-176.537,8.151,148.584
C00901=1176.034,324.381,-73.758,-176.539,8.148,148.584
C00902=1176.038,324.134,-73.726,-176.541,8.145,148.583
C00903=1176.043,323.885,-73.694,-176.544,8.142,148.583
C00904=1176.047,323.637,-73.663,-176.546,8.138,148.583
C00905=1176.051,323.389,-73.631,-176.549,8.135,148.583
C00906=1176.054,323.141,-73.599,-176.552,8.131,148.583
C00907=1176.060,322.894,-73.567,-176.554,8.128,148.583
C00908=1176.063,322.646,-73.535,-176.557,8.125,148.583
C00909=1176.067,322.397,-73.504,-176.559,8.122,148.583
C00910=1176.072,322.150,-73.473,-176.562,8.119,148.583
C00911=1176.075,321.902,-73.441,-176.564,8.116,148.583
C00912=1176.080,321.654,-73.409,-176.567,8.112,148.582
C00913=1176.084,321.406,-73.377,-176.569,8.109,148.582
C00914=1176.088,321.157,-73.346,-176.572,8.106,148.582
C00915=1176.092,320.910,-73.314,-176.574,8.103,148.582
C00916=1176.096,320.662,-73.282,-176.577,8.100,148.582
C00917=1176.101,320.414,-73.252,-176.579,8.097,148.582
C00918=1176.104,320.166,-73.220,-176.582,8.093,148.582
C00919=1176.109,319.918,-73.188,-176.584,8.090,148.582
C00920=1176.113,319.670,-73.157,-176.587,8.087,148.582
C00921=1176.118,319.422,-73.125,-176.589,8.084,148.582
C00922=1176.121,319.174,-73.093,-176.592,8.081,148.581
C00923=1176.125,318.926,-73.062,-176.594,8.078,148.581
C00924=1176.130,318.678,-73.031,-176.597,8.074,148.581
C00925=1176.134,318.430,-73.000,-176.599,8.072,148.581
C00926=1176.138,318.182,-72.968,-176.602,8.068,148.581
C00927=1176.142,317.934,-72.936,-176.604,8.065,148.581
C00928=1176.146,317.686,-72.906,-176.607,8.062,148.581
C00929=1176.150,317.438,-72.874,-176.609,8.059,148.581
C00930=1176.155,317.190,-72.843,-176.612,8.056,148.581
C00931=1176.158,316.942,-72.811,-176.614,8.053,148.581
C00932=1176.163,316.694,-72.780,-176.617,8.049,148.580
C00933=1176.167,316.446,-72.748,-176.619,8.046,148.580
C00934=1176.171,316.198,-72.718,-176.622,8.043,148.581
C00935=1176.175,315.950,-72.686,-176.624,8.041,148.580
C00936=1176.180,315.702,-72.655,-176.626,8.038,148.580
C00937=1176.184,315.454,-72.624,-176.629,8.035,148.580
C00938=1176.188,315.206,-72.592,-176.631,8.032,148.580
C00939=1176.193,314.958,-72.562,-176.634,8.028,148.580
C00940=1176.196,314.710,-72.530,-176.636,8.025,148.580
C00941=1176.202,314.433,-72.495,-176.640,8.021,148.580
C00942=1176.206,314.156,-72.461,-176.642,8.018,148.580
C00943=1176.211,313.879,-72.425,-176.645,8.014,148.580
C00944=1176.215,313.603,-72.391,-176.648,8.011,148.580
C00945=1176.219,313.355,-72.360,-176.650,8.008,148.580
C00946=1176.224,313.107,-72.329,-176.653,8.005,148.580
C00947=1176.228,312.858,-72.298,-176.655,8.002,148.579
C00948=1176.232,312.611,-72.267,-176.658,7.999,148.579
C00949=1176.236,312.362,-72.236,-176.661,7.996,148.579
C00950=1176.241,312.114,-72.205,-176.663,7.992,148.579
C00951=1176.246,311.866,-72.174,-176.666,7.989,148.579
C00952=1176.249,311.619,-72.143,-176.669,7.987,148.579
C00953=1176.253,311.371,-72.112,-176.671,7.983,148.579
C00954=1176.258,311.123,-72.081,-176.674,7.980,148.579
C00955=1176.262,310.874,-72.050,-176.676,7.977,148.579
C00956=1176.266,310.626,-72.019,-176.679,7.974,148.579
C00957=1176.270,310.378,-71.987,-176.681,7.971,148.579
C00958=1176.274,310.131,-71.957,-176.684,7.968,148.579
C00959=1176.279,309.883,-71.927,-176.686,7.965,148.579
C00960=1176.283,309.634,-71.895,-176.689,7.962,148.579
C00961=1176.287,309.386,-71.865,-176.691,7.959,148.579
C00962=1176.291,309.138,-71.834,-176.693,7.956,148.579
C00963=1176.295,308.890,-71.803,-176.696,7.953,148.578
C00964=1176.300,308.642,-71.773,-176.698,7.950,148.578
C00965=1176.304,308.394,-71.742,-176.701,7.947,148.578
C00966=1176.308,308.146,-71.712,-176.703,7.944,148.578
C00967=1176.312,307.897,-71.681,-176.706,7.941,148.578
C00968=1176.317,307.649,-71.650,-176.709,7.938,148.578
C00969=1176.321,307.402,-71.619,-176.711,7.934,148.578
C00970=1176.325,307.153,-71.588,-176.714,7.931,148.578
C00971=1176.329,306.905,-71.558,-176.717,7.928,148.578
C00972=1176.334,306.657,-71.527,-176.719,7.925,148.578
C00973=1176.338,306.410,-71.497,-176.722,7.922,148.578
C00974=1176.342,306.161,-71.466,-176.724,7.919,148.578
C00975=1176.346,305.913,-71.435,-176.727,7.916,148.578
C00976=1176.350,305.665,-71.405,-176.729,7.913,148.578
C00977=1176.355,305.417,-71.374,-176.732,7.910,148.578
C00978=1176.359,305.169,-71.343,-176.735,7.907,148.578
C00979=1176.363,304.920,-71.313,-176.736,7.904,148.578
C00980=1176.368,304.672,-71.283,-176.739,7.901,148.578
C00981=1176.372,304.425,-71.252,-176.742,7.898,148.578
C00982=1176.376,304.176,-71.221,-176.744,7.895,148.578
C00983=1176.380,303.928,-71.191,-176.747,7.892,148.578
C00984=1176.384,303.681,-71.160,-176.750,7.889,148.578
C00985=1176.389,303.432,-71.130,-176.752,7.886,148.578
C00986=1176.393,303.184,-71.100,-176.755,7.883,148.577
C00987=1176.397,302.936,-71.069,-176.757,7.880,148.577
C00988=1176.402,302.688,-71.038,-176.760,7.877,148.578
C00989=1176.406,302.439,-71.009,-176.762,7.874,148.577
C00990=1176.410,302.192,-70.978,-176.765,7.871,148.577
C00991=1176.414,301.944,-70.948,-176.768,7.868,148.577
C00992=1176.419,301.695,-70.918,-176.770,7.865,148.577
C00993=1176.422,301.447,-70.887,-176.772,7.862,148.577
C00994=1176.427,301.199,-70.857,-176.775,7.859,148.577
C00995=1176.431,300.951,-70.827,-176.778,7.856,148.577
C00996=1176.436,300.703,-70.796,-176.780,7.853,148.577
C00997=1176.440,300.455,-70.766,-176.783,7.850,148.577
C00998=1176.445,300.207,-70.736,-176.785,7.847,148.577
C00999=1176.448,299.958,-70.706,-176.788,7.844,148.577
C01000=1176.452,299.710,-70.676,-176.791,7.841,148.577
C01001=1176.457,299.462,-70.645,-176.793,7.838,148.577
C01002=1176.461,299.214,-70.615,-176.796,7.835,148.577
C01003=1176.465,298.966,-70.585,-176.798,7.832,148.577
C01004=1176.469,298.718,-70.555,-176.801,7.829,148.577
C01005=1176.474,298.470,-70.525,-176.803,7.826,148.577
C01006=1176.478,298.222,-70.495,-176.806,7.823,148.577
C01007=1176.482,297.974,-70.465,-176.809,7.820,148.577
C01008=1176.486,297.725,-70.434,-176.811,7.817,148.577
C01009=1176.491,297.477,-70.405,-176.814,7.814,148.577
C01010=1176.494,297.229,-70.375,-176.816,7.811,148.577
C01011=1176.499,296.980,-70.344,-176.819,7.808,148.577
C01012=1176.503,296.732,-70.315,-176.821,7.806,148.577
C01013=1176.507,296.485,-70.285,-176.824,7.803,148.577
C01014=1176.512,296.236,-70.255,-176.826,7.799,148.577
C01015=1176.516,295.988,-70.225,-176.829,7.796,148.577
C01016=1176.520,295.740,-70.195,-176.832,7.793,148.577
C01017=1176.525,295.491,-70.165,-176.834,7.790,148.577
C01018=1176.529,295.244,-70.135,-176.837,7.787,148.577
C01019=1176.533,294.996,-70.106,-176.839,7.784,148.577
C01020=1176.538,294.747,-70.075,-176.842,7.781,148.577
C01021=1176.542,294.499,-70.045,-176.844,7.779,148.577
C01022=1176.546,294.251,-70.016,-176.847,7.776,148.577
C01023=1176.550,294.003,-69.986,-176.850,7.773,148.577
C01024=1176.554,293.755,-69.956,-176.852,7.770,148.577
C01025=1176.559,293.507,-69.926,-176.855,7.767,148.577
C01026=1176.563,293.258,-69.897,-176.857,7.764,148.577
C01027=1176.568,293.010,-69.867,-176.860,7.761,148.577
C01028=1176.572,292.762,-69.838,-176.863,7.758,148.577
C01029=1176.576,292.514,-69.807,-176.865,7.756,148.577
C01030=1176.581,292.266,-69.778,-176.867,7.752,148.577
C01031=1176.585,292.017,-69.748,-176.870,7.749,148.577
C01032=1176.589,291.769,-69.719,-176.873,7.746,148.577
C01033=1176.593,291.521,-69.689,-176.876,7.743,148.577
C01034=1176.597,291.272,-69.660,-176.878,7.740,148.577
C01035=1176.602,291.024,-69.629,-176.881,7.737,148.577
C01036=1176.606,290.776,-69.600,-176.883,7.735,148.577
C01037=1176.610,290.528,-69.570,-176.885,7.732,148.577
C01038=1176.614,290.280,-69.541,-176.888,7.729,148.577
C01039=1176.619,290.031,-69.511,-176.891,7.726,148.577
C01040=1176.623,289.783,-69.482,-176.894,7.723,148.577
C01041=1176.627,289.535,-69.452,-176.896,7.720,148.577
C01042=1176.631,289.287,-69.423,-176.899,7.717,148.577
C01043=1176.635,289.038,-69.393,-176.901,7.715,148.577
C01044=1176.640,288.790,-69.364,-176.904,7.712,148.577
C01045=1176.645,288.516,-69.331,-176.907,7.708,148.577
C01046=1176.650,288.241,-69.298,-176.910,7.705,148.577
C01047=1176.654,287.966,-69.266,-176.912,7.702,148.577
C01048=1176.659,287.692,-69.233,-176.915,7.699,148.577
C01049=1176.663,287.443,-69.204,-176.918,7.696,148.577
C01050=1176.668,287.195,-69.175,-176.921,7.693,148.577
C01051=1176.672,286.947,-69.145,-176.923,7.690,148.577
C01052=1176.676,286.698,-69.116,-176.926,7.687,148.577
C01053=1176.680,286.450,-69.087,-176.928,7.684,148.577
C01054=1176.685,286.202,-69.058,-176.930,7.682,148.577
C01055=1176.689,285.954,-69.028,-176.933,7.679,148.577
C01056=1176.694,285.705,-68.999,-176.936,7.676,148.577
C01057=1176.698,285.457,-68.969,-176.939,7.673,148.577
C01058=1176.702,285.209,-68.940,-176.941,7.670,148.577
C01059=1176.706,284.960,-68.911,-176.944,7.667,148.577
C01060=1176.711,284.712,-68.882,-176.946,7.664,148.577
C01061=1176.715,284.464,-68.853,-176.949,7.661,148.577
C01062=1176.720,284.216,-68.823,-176.952,7.658,148.577
C01063=1176.724,283.968,-68.794,-176.954,7.655,148.577
C01064=1176.727,283.719,-68.766,-176.957,7.652,148.577
C01065=1176.732,283.472,-68.737,-176.959,7.650,148.577
C01066=1176.736,283.223,-68.707,-176.962,7.647,148.577
C01067=1176.741,282.974,-68.678,-176.964,7.644,148.577
C01068=1176.745,282.726,-68.649,-176.967,7.641,148.577
C01069=1176.749,282.478,-68.619,-176.970,7.638,148.577
C01070=1176.754,282.230,-68.591,-176.972,7.636,148.577
C01071=1176.759,281.981,-68.562,-176.975,7.633,148.577
C01072=1176.762,281.733,-68.533,-176.977,7.630,148.577
C01073=1176.767,281.485,-68.504,-176.980,7.627,148.578
C01074=1176.771,281.237,-68.475,-176.983,7.624,148.578
C01075=1176.775,280.989,-68.446,-176.986,7.621,148.578
C01076=1176.780,280.740,-68.417,-176.988,7.619,148.578
C01077=1176.783,280.492,-68.388,-176.991,7.616,148.578
C01078=1176.788,280.244,-68.360,-176.993,7.613,148.578
C01079=1176.793,279.995,-68.330,-176.996,7.610,148.578
C01080=1176.797,279.747,-68.301,-176.998,7.607,148.578
C01081=1176.801,279.498,-68.272,-177.001,7.605,148.578
C01082=1176.806,279.250,-68.244,-177.003,7.602,148.578
C01083=1176.810,279.002,-68.215,-177.006,7.599,148.578
C01084=1176.814,278.753,-68.186,-177.009,7.596,148.578
C01085=1176.818,278.506,-68.157,-177.011,7.593,148.578
C01086=1176.823,278.257,-68.129,-177.014,7.590,148.578
C01087=1176.827,278.009,-68.099,-177.016,7.587,148.578
C01088=1176.832,277.761,-68.071,-177.019,7.584,148.578
C01089=1176.836,277.513,-68.042,-177.022,7.582,148.578
C01090=1176.840,277.264,-68.013,-177.024,7.579,148.578
C01091=1176.845,277.016,-67.985,-177.027,7.576,148.578
C01092=1176.849,276.768,-67.956,-177.029,7.573,148.578
C01093=1176.853,276.519,-67.927,-177.032,7.570,148.578
C01094=1176.858,276.271,-67.899,-177.035,7.567,148.578
C01095=1176.862,276.023,-67.870,-177.037,7.565,148.578
C01096=1176.866,275.774,-67.841,-177.040,7.562,148.578
C01097=1176.870,275.526,-67.814,-177.043,7.559,148.578
C01098=1176.875,275.278,-67.784,-177.045,7.556,148.579
C01099=1176.879,275.029,-67.755,-177.047,7.554,148.579
C01100=1176.884,274.781,-67.728,-177.050,7.551,148.579
C01101=1176.888,274.533,-67.698,-177.053,7.548,148.579
C01102=1176.892,274.285,-67.670,-177.056,7.545,148.579
C01103=1176.897,274.036,-67.642,-177.058,7.543,148.579
C01104=1176.901,273.787,-67.613,-177.061,7.540,148.579
C01105=1176.905,273.539,-67.585,-177.063,7.537,148.579
C01106=1176.910,273.291,-67.556,-177.066,7.534,148.579
C01107=1176.914,273.043,-67.528,-177.068,7.532,148.579
C01108=1176.918,272.794,-67.499,-177.071,7.529,148.579
C01109=1176.922,272.545,-67.471,-177.074,7.526,148.579
C01110=1176.927,272.297,-67.443,-177.076,7.523,148.579
C01111=1176.931,272.049,-67.414,-177.079,7.520,148.579
C01112=1176.936,271.801,-67.385,-177.081,7.518,148.579
C01113=1176.940,271.553,-67.357,-177.084,7.515,148.579
C01114=1176.945,271.304,-67.329,-177.087,7.512,148.579
C01115=1176.948,271.056,-67.301,-177.089,7.510,148.579
C01116=1176.953,270.807,-67.272,-177.092,7.507,148.580
C01117=1176.957,270.559,-67.244,-177.094,7.504,148.580
C01118=1176.962,270.310,-67.215,-177.097,7.501,148.580
C01119=1176.966,270.062,-67.188,-177.100,7.499,148.580
C01120=1176.970,269.814,-67.160,-177.103,7.496,148.580
C01121=1176.975,269.565,-67.131,-177.105,7.493,148.580
C01122=1176.979,269.317,-67.103,-177.108,7.490,148.580
C01123=1176.984,269.069,-67.075,-177.110,7.488,148.580
C01124=1176.987,268.820,-67.047,-177.113,7.485,148.580
C01125=1176.993,268.572,-67.018,-177.116,7.482,148.580
C01126=1176.996,268.323,-66.990,-177.118,7.479,148.580
C01127=1177.001,268.075,-66.962,-177.121,7.477,148.580
C01128=1177.005,267.827,-66.934,-177.123,7.474,148.580
C01129=1177.009,267.579,-66.906,-177.126,7.471,148.580
C01130=1177.013,267.330,-66.878,-177.128,7.469,148.581
C01131=1177.019,267.081,-66.850,-177.131,7.466,148.581
C01132=1177.023,266.833,-66.822,-177.134,7.463,148.581
C01133=1177.027,266.585,-66.794,-177.136,7.460,148.581
C01134=1177.032,266.337,-66.766,-177.139,7.458,148.581
C01135=1177.036,266.088,-66.737,-177.142,7.455,148.581
C01136=1177.040,265.840,-66.710,-177.145,7.452,148.581
C01137=1177.045,265.591,-66.682,-177.147,7.450,148.581
C01138=1177.049,265.343,-66.654,-177.150,7.447,148.581
C01139=1177.053,265.095,-66.626,-177.152,7.444,148.581
C01140=1177.057,264.846,-66.598,-177.155,7.441,148.581
C01141=1177.063,264.598,-66.570,-177.157,7.439,148.581
C01142=1177.066,264.349,-66.542,-177.160,7.436,148.581
C01143=1177.071,264.101,-66.514,-177.163,7.433,148.582
C01144=1177.075,263.853,-66.487,-177.165,7.431,148.582
C01145=1177.080,263.604,-66.459,-177.168,7.428,148.582
C01146=1177.084,263.356,-66.431,-177.171,7.425,148.582
C01147=1177.088,263.107,-66.403,-177.173,7.423,148.582
C01148=1177.093,262.859,-66.376,-177.176,7.420,148.582
C01149=1177.097,262.585,-66.345,-177.178,7.417,148.582
C01150=1177.102,262.313,-66.315,-177.182,7.414,148.582
C01151=1177.107,262.040,-66.284,-177.184,7.411,148.582
C01152=1177.112,261.767,-66.254,-177.187,7.408,148.582
C01153=1177.116,261.518,-66.226,-177.190,7.406,148.583
C01154=1177.121,261.270,-66.198,-177.193,7.403,148.583
C01155=1177.125,261.021,-66.170,-177.195,7.401,148.583
C01156=1177.129,260.773,-66.143,-177.198,7.398,148.583
C01157=1177.134,260.525,-66.115,-177.201,7.395,148.583
C01158=1177.138,260.276,-66.087,-177.203,7.393,148.583
C01159=1177.143,260.028,-66.060,-177.206,7.390,148.583
C01160=1177.147,259.780,-66.032,-177.208,7.387,148.583
C01161=1177.152,259.531,-66.005,-177.211,7.385,148.583
C01162=1177.155,259.283,-65.977,-177.214,7.382,148.584
C01163=1177.160,259.034,-65.950,-177.216,7.379,148.584
C01164=1177.164,258.786,-65.922,-177.219,7.377,148.584
C01165=1177.169,258.537,-65.894,-177.221,7.374,148.584
C01166=1177.173,258.289,-65.867,-177.224,7.371,148.584
C01167=1177.178,258.041,-65.840,-177.226,7.369,148.584
C01168=1177.182,257.791,-65.812,-177.230,7.366,148.584
C01169=1177.186,257.544,-65.784,-177.232,7.363,148.584
C01170=1177.191,257.295,-65.757,-177.234,7.361,148.584
C01171=1177.195,257.047,-65.730,-177.237,7.358,148.584
C01172=1177.199,256.798,-65.702,-177.240,7.355,148.584
C01173=1177.204,256.549,-65.675,-177.243,7.353,148.585
C01174=1177.208,256.302,-65.647,-177.245,7.350,148.585
C01175=1177.213,256.053,-65.620,-177.248,7.347,148.585
C01176=1177.217,255.804,-65.593,-177.250,7.345,148.585
C01177=1177.221,255.555,-65.566,-177.253,7.342,148.585
C01178=1177.226,255.308,-65.538,-177.256,7.339,148.585
C01179=1177.230,255.059,-65.511,-177.258,7.337,148.585
C01180=1177.235,254.811,-65.484,-177.261,7.334,148.585
C01181=1177.239,254.561,-65.456,-177.263,7.332,148.586
C01182=1177.243,254.313,-65.429,-177.266,7.329,148.586
C01183=1177.248,254.065,-65.402,-177.269,7.327,148.586
C01184=1177.253,253.816,-65.375,-177.271,7.324,148.586
C01185=1177.257,253.568,-65.347,-177.274,7.321,148.586
C01186=1177.261,253.319,-65.320,-177.277,7.318,148.586
C01187=1177.265,253.071,-65.293,-177.279,7.317,148.586
C01188=1177.270,252.823,-65.266,-177.282,7.314,148.586
C01189=1177.274,252.574,-65.239,-177.284,7.312,148.587
C01190=1177.279,252.326,-65.212,-177.287,7.309,148.587
C01191=1177.284,252.077,-65.185,-177.290,7.306,148.587
C01192=1177.288,251.828,-65.157,-177.293,7.304,148.587
C01193=1177.292,251.580,-65.131,-177.295,7.301,148.587
C01194=1177.296,251.331,-65.104,-177.298,7.298,148.587
C01195=1177.301,251.083,-65.077,-177.300,7.296,148.587
C01196=1177.305,250.835,-65.049,-177.303,7.293,148.587
C01197=1177.310,250.587,-65.022,-177.306,7.291,148.588
C01198=1177.314,250.338,-64.995,-177.308,7.288,148.588
C01199=1177.318,250.089,-64.968,-177.311,7.285,148.588
C01200=1177.323,249.841,-64.941,-177.314,7.283,148.588
C01201=1177.327,249.592,-64.914,-177.316,7.280,148.588
C01202=1177.332,249.344,-64.887,-177.319,7.278,148.588
C01203=1177.336,249.095,-64.860,-177.322,7.275,148.588
C01204=1177.341,248.846,-64.834,-177.325,7.272,148.589
C01205=1177.346,248.598,-64.807,-177.327,7.270,148.589
C01206=1177.349,248.350,-64.780,-177.330,7.267,148.589
C01207=1177.354,248.101,-64.753,-177.332,7.265,148.589
C01208=1177.359,247.853,-64.726,-177.335,7.263,148.589
C01209=1177.363,247.604,-64.699,-177.338,7.260,148.589
C01210=1177.367,247.355,-64.672,-177.340,7.258,148.589
C01211=1177.371,247.107,-64.645,-177.343,7.255,148.590
C01212=1177.376,246.858,-64.618,-177.345,7.253,148.590
C01213=1177.380,246.609,-64.592,-177.348,7.250,148.590
C01214=1177.385,246.361,-64.565,-177.351,7.248,148.590
C01215=1177.390,246.112,-64.538,-177.353,7.245,148.590
C01216=1177.393,245.864,-64.512,-177.356,7.242,148.590
C01217=1177.398,245.616,-64.485,-177.359,7.240,148.590
C01218=1177.402,245.367,-64.459,-177.361,7.237,148.590
C01219=1177.407,245.119,-64.432,-177.364,7.235,148.591
C01220=1177.412,244.870,-64.405,-177.367,7.232,148.591
C01221=1177.416,244.622,-64.378,-177.369,7.230,148.591
C01222=1177.421,244.373,-64.352,-177.372,7.227,148.591
C01223=1177.424,244.125,-64.326,-177.375,7.225,148.591
C01224=1177.429,243.876,-64.299,-177.377,7.222,148.591
C01225=1177.434,243.628,-64.272,-177.380,7.219,148.591
C01226=1177.438,243.379,-64.246,-177.383,7.218,148.592
C01227=1177.443,243.130,-64.219,-177.385,7.215,148.592
C01228=1177.447,242.882,-64.192,-177.388,7.213,148.592
C01229=1177.452,242.633,-64.166,-177.391,7.210,148.592
C01230=1177.455,242.385,-64.139,-177.393,7.208,148.592
C01231=1177.460,242.136,-64.113,-177.396,7.205,148.592
C01232=1177.464,241.887,-64.087,-177.399,7.202,148.593
C01233=1177.469,241.639,-64.060,-177.401,7.200,148.593
C01234=1177.473,241.390,-64.034,-177.404,7.197,148.593
C01235=1177.478,241.142,-64.007,-177.406,7.195,148.593
C01236=1177.483,240.894,-63.981,-177.409,7.192,148.593
C01237=1177.487,240.645,-63.954,-177.411,7.190,148.593
C01238=1177.492,240.396,-63.929,-177.415,7.188,148.594
C01239=1177.496,240.148,-63.901,-177.417,7.185,148.594
C01240=1177.500,239.899,-63.876,-177.420,7.182,148.594
C01241=1177.505,239.650,-63.849,-177.422,7.181,148.594
C01242=1177.509,239.402,-63.823,-177.425,7.178,148.594
C01243=1177.513,239.153,-63.796,-177.428,7.176,148.595
C01244=1177.518,238.904,-63.770,-177.430,7.173,148.595
C01245=1177.522,238.656,-63.744,-177.432,7.171,148.595
C01246=1177.528,238.408,-63.718,-177.436,7.168,148.595
C01247=1177.532,238.160,-63.691,-177.438,7.166,148.595
C01248=1177.536,237.911,-63.665,-177.441,7.163,148.595
C01249=1177.541,237.662,-63.639,-177.444,7.160,148.595
C01250=1177.545,237.413,-63.613,-177.446,7.158,148.596
C01251=1177.549,237.165,-63.587,-177.449,7.156,148.596
C01252=1177.554,236.916,-63.561,-177.451,7.153,148.596
C01253=1177.559,236.645,-63.532,-177.455,7.151,148.596
C01254=1177.564,236.373,-63.504,-177.457,7.148,148.596
C01255=1177.569,236.101,-63.475,-177.461,7.145,148.597
C01256=1177.573,235.830,-63.447,-177.463,7.143,148.597
C01257=1177.577,235.581,-63.420,-177.466,7.140,148.597
C01258=1177.582,235.332,-63.394,-177.468,7.138,148.597
C01259=1177.587,235.084,-63.369,-177.471,7.136,148.597
C01260=1177.591,234.835,-63.343,-177.474,7.133,148.598
C01261=1177.595,234.587,-63.316,-177.476,7.131,148.598
C01262=1177.600,234.338,-63.290,-177.479,7.129,148.598
C01263=1177.604,234.089,-63.264,-177.482,7.126,148.598
C01264=1177.609,233.841,-63.239,-177.484,7.124,148.598
C01265=1177.613,233.593,-63.212,-177.487,7.121,148.598
C01266=1177.618,233.344,-63.186,-177.490,7.119,148.599
C01267=1177.622,233.095,-63.160,-177.493,7.116,148.599
C01268=1177.627,232.846,-63.134,-177.495,7.114,148.599
C01269=1177.631,232.598,-63.109,-177.498,7.111,148.599
C01270=1177.636,232.349,-63.083,-177.500,7.109,148.599
C01271=1177.641,232.100,-63.057,-177.503,7.107,148.600
C01272=1177.645,231.852,-63.031,-177.506,7.105,148.600
C01273=1177.649,231.604,-63.005,-177.509,7.102,148.600
C01274=1177.654,231.355,-62.979,-177.511,7.100,148.600
C01275=1177.658,231.106,-62.954,-177.514,7.097,148.600
C01276=1177.663,230.857,-62.927,-177.516,7.095,148.600
C01277=1177.668,230.609,-62.902,-177.519,7.093,148.601
C01278=1177.672,230.360,-62.876,-177.522,7.090,148.601
C01279=1177.676,230.112,-62.850,-177.524,7.088,148.601
C01280=1177.681,229.863,-62.825,-177.527,7.085,148.601
C01281=1177.685,229.615,-62.799,-177.530,7.084,148.602
C01282=1177.689,229.366,-62.774,-177.533,7.081,148.602
C01283=1177.694,229.117,-62.748,-177.535,7.079,148.602
C01284=1177.698,228.869,-62.722,-177.538,7.076,148.602
C01285=1177.703,228.620,-62.696,-177.540,7.074,148.602
C01286=1177.708,228.371,-62.670,-177.543,7.071,148.603
C01287=1177.712,228.123,-62.645,-177.546,7.069,148.603
C01288=1177.717,227.874,-62.619,-177.548,7.067,148.603
C01289=1177.721,227.625,-62.594,-177.551,7.064,148.603
C01290=1177.726,227.377,-62.569,-177.554,7.062,148.603
C01291=1177.730,227.128,-62.543,-177.556,7.059,148.603
C01292=1177.734,226.879,-62.517,-177.559,7.058,148.604
C01293=1177.739,226.631,-62.492,-177.562,7.055,148.604
C01294=1177.743,226.382,-62.466,-177.564,7.053,148.604
C01295=1177.748,226.133,-62.440,-177.568,7.050,148.604
C01296=1177.753,225.884,-62.416,-177.570,7.048,148.605
C01297=1177.757,225.636,-62.390,-177.572,7.046,148.605
C01298=1177.762,225.388,-62.365,-177.575,7.043,148.605
C01299=1177.766,225.139,-62.339,-177.578,7.042,148.605
C01300=1177.770,224.890,-62.313,-177.581,7.039,148.605
C01301=1177.775,224.641,-62.288,-177.583,7.037,148.606
C01302=1177.780,224.392,-62.263,-177.585,7.035,148.606
C01303=1177.785,224.144,-62.237,-177.589,7.032,148.606
C01304=1177.788,223.895,-62.213,-177.591,7.030,148.606
C01305=1177.793,223.646,-62.187,-177.594,7.027,148.607
C01306=1177.797,223.398,-62.162,-177.596,7.025,148.607
C01307=1177.802,223.150,-62.136,-177.599,7.023,148.607
C01308=1177.807,222.901,-62.111,-177.602,7.020,148.607
C01309=1177.811,222.652,-62.086,-177.604,7.019,148.607
C01310=1177.815,222.403,-62.060,-177.608,7.016,148.608
C01311=1177.820,222.154,-62.035,-177.610,7.014,148.608
C01312=1177.825,221.906,-62.009,-177.613,7.011,148.608
C01313=1177.829,221.657,-61.985,-177.615,7.009,148.608
C01314=1177.833,221.408,-61.960,-177.618,7.007,148.609
C01315=1177.838,221.160,-61.934,-177.621,7.004,148.609
C01316=1177.843,220.911,-61.909,-177.623,7.003,148.609
C01317=1177.847,220.663,-61.884,-177.626,7.000,148.609
C01318=1177.852,220.413,-61.859,-177.629,6.998,148.609
C01319=1177.856,220.166,-61.834,-177.631,6.996,148.610
C01320=1177.860,219.916,-61.809,-177.634,6.993,148.610
C01321=1177.865,219.668,-61.783,-177.637,6.991,148.610
C01322=1177.870,219.419,-61.758,-177.639,6.989,148.610
C01323=1177.874,219.171,-61.734,-177.642,6.986,148.611
C01324=1177.878,218.921,-61.709,-177.644,6.984,148.611
C01325=1177.883,218.673,-61.683,-177.648,6.982,148.611
C01326=1177.888,218.424,-61.658,-177.650,6.980,148.611
C01327=1177.892,218.176,-61.633,-177.652,6.978,148.611
C01328=1177.896,217.927,-61.608,-177.656,6.975,148.612
C01329=1177.902,217.678,-61.584,-177.658,6.973,148.612
C01330=1177.906,217.429,-61.558,-177.661,6.970,148.612
C01331=1177.910,217.181,-61.534,-177.664,6.969,148.613
C01332=1177.914,216.932,-61.508,-177.666,6.966,148.613
C01333=1177.920,216.683,-61.483,-177.669,6.964,148.613
C01334=1177.923,216.434,-61.459,-177.671,6.962,148.613
C01335=1177.928,216.186,-61.434,-177.674,6.960,148.613
C01336=1177.933,215.937,-61.409,-177.677,6.957,148.614
C01337=1177.937,215.688,-61.384,-177.679,6.955,148.614
C01338=1177.942,215.440,-61.359,-177.682,6.953,148.614
C01339=1177.946,215.191,-61.334,-177.685,6.950,148.614
C01340=1177.951,214.942,-61.310,-177.687,6.949,148.615
C01341=1177.955,214.693,-61.284,-177.690,6.947,148.615
C01342=1177.960,214.445,-61.260,-177.693,6.944,148.615
C01343=1177.965,214.196,-61.236,-177.695,6.942,148.615
C01344=1177.969,213.947,-61.210,-177.699,6.939,148.616
C01345=1177.974,213.698,-61.186,-177.701,6.937,148.616
C01346=1177.978,213.450,-61.161,-177.704,6.935,148.616
C01347=1177.982,213.201,-61.137,-177.706,6.933,148.616
C01348=1177.987,212.952,-61.112,-177.709,6.931,148.617
C01349=1177.992,212.703,-61.087,-177.712,6.929,148.617
C01350=1177.996,212.455,-61.063,-177.714,6.926,148.617
C01351=1178.001,212.207,-61.037,-177.717,6.924,148.617
C01352=1178.005,211.957,-61.013,-177.720,6.922,148.618
C01353=1178.010,211.709,-60.988,-177.722,6.919,148.618
C01354=1178.014,211.460,-60.964,-177.725,6.918,148.618
C01355=1178.019,211.211,-60.939,-177.728,6.916,148.618
C01356=1178.023,210.962,-60.915,-177.731,6.913,148.619
C01357=1178.028,210.692,-60.888,-177.733,6.911,148.619
C01358=1178.033,210.421,-60.861,-177.736,6.908,148.619
C01359=1178.038,210.151,-60.835,-177.739,6.907,148.619
C01360=1178.043,209.881,-60.808,-177.742,6.904,148.620
C01361=1178.047,209.632,-60.783,-177.745,6.902,148.620
C01362=1178.052,209.383,-60.759,-177.748,6.899,148.620
C01363=1178.057,209.135,-60.735,-177.750,6.897,148.620
C01364=1178.061,208.885,-60.710,-177.753,6.895,148.621
C01365=1178.066,208.637,-60.686,-177.756,6.893,148.621
C01366=1178.071,208.388,-60.661,-177.758,6.891,148.621
C01367=1178.075,208.139,-60.638,-177.761,6.889,148.621
C01368=1178.080,207.890,-60.613,-177.763,6.887,148.622
C01369=1178.084,207.641,-60.588,-177.766,6.884,148.622
C01370=1178.089,207.393,-60.564,-177.769,6.882,148.622
C01371=1178.094,207.144,-60.540,-177.771,6.880,148.623
C01372=1178.098,206.895,-60.515,-177.774,6.878,148.623
C01373=1178.103,206.646,-60.491,-177.777,6.876,148.623
C01374=1178.107,206.398,-60.467,-177.780,6.874,148.623
C01375=1178.112,206.150,-60.442,-177.783,6.871,148.624
C01376=1178.116,205.900,-60.417,-177.785,6.869,148.624
C01377=1178.121,205.651,-60.394,-177.788,6.867,148.624
C01378=1178.125,205.403,-60.370,-177.790,6.866,148.624
C01379=1178.130,205.154,-60.345,-177.793,6.863,148.625
C01380=1178.134,204.905,-60.321,-177.796,6.861,148.625
C01381=1178.138,204.656,-60.297,-177.798,6.859,148.625
C01382=1178.144,204.407,-60.273,-177.801,6.856,148.625
C01383=1178.148,204.159,-60.249,-177.804,6.854,148.626
C01384=1178.153,203.910,-60.225,-177.806,6.853,148.626
C01385=1178.156,203.661,-60.200,-177.809,6.850,148.626
C01386=1178.162,203.412,-60.176,-177.812,6.848,148.627
C01387=1178.166,203.163,-60.152,-177.815,6.846,148.627
C01388=1178.171,202.915,-60.128,-177.817,6.844,148.627
C01389=1178.175,202.667,-60.104,-177.819,6.842,148.627
C01390=1178.180,202.417,-60.080,-177.823,6.839,148.628
C01391=1178.184,202.168,-60.056,-177.825,6.838,148.628
C01392=1178.189,201.920,-60.032,-177.828,6.836,148.628
C01393=1178.193,201.671,-60.008,-177.831,6.833,148.628
C01394=1178.199,201.422,-59.984,-177.833,6.831,148.629
C01395=1178.203,201.174,-59.960,-177.836,6.829,148.629
C01396=1178.208,200.925,-59.936,-177.838,6.827,148.629
C01397=1178.211,200.675,-59.912,-177.842,6.825,148.630
C01398=1178.216,200.426,-59.888,-177.844,6.823,148.630
C01399=1178.221,200.178,-59.864,-177.847,6.821,148.630
C01400=1178.226,199.929,-59.840,-177.849,6.819,148.630
C01401=1178.230,199.680,-59.816,-177.852,6.816,148.631
C01402=1178.235,199.432,-59.792,-177.855,6.815,148.631
C01403=1178.239,199.183,-59.769,-177.857,6.812,148.631
C01404=1178.244,198.934,-59.745,-177.860,6.811,148.632
C01405=1178.249,198.685,-59.721,-177.863,6.808,148.632
C01406=1178.252,198.436,-59.697,-177.866,6.806,148.632
C01407=1178.258,198.187,-59.673,-177.868,6.804,148.632
C01408=1178.262,197.938,-59.649,-177.871,6.802,148.633
C01409=1178.267,197.689,-59.626,-177.873,6.801,148.633
C01410=1178.271,197.441,-59.601,-177.876,6.798,148.633
C01411=1178.276,197.192,-59.578,-177.879,6.796,148.633
C01412=1178.281,196.943,-59.555,-177.881,6.794,148.634
C01413=1178.285,196.695,-59.531,-177.884,6.792,148.634
C01414=1178.290,196.446,-59.507,-177.887,6.790,148.634
C01415=1178.294,196.197,-59.483,-177.890,6.788,148.635
C01416=1178.299,195.948,-59.460,-177.892,6.786,148.635
C01417=1178.304,195.699,-59.437,-177.895,6.784,148.635
C01418=1178.308,195.451,-59.412,-177.898,6.781,148.636
C01419=1178.313,195.202,-59.389,-177.901,6.780,148.636
C01420=1178.317,194.953,-59.366,-177.903,6.777,148.636
C01421=1178.322,194.704,-59.342,-177.906,6.776,148.636
C01422=1178.326,194.455,-59.318,-177.908,6.774,148.637
C01423=1178.331,194.206,-59.295,-177.911,6.771,148.637
C01424=1178.336,193.958,-59.271,-177.914,6.769,148.637
C01425=1178.340,193.709,-59.248,-177.916,6.767,148.638
C01426=1178.345,193.460,-59.224,-177.919,6.766,148.638
C01427=1178.350,193.211,-59.201,-177.922,6.764,148.638
C01428=1178.354,192.962,-59.177,-177.925,6.761,148.639
C01429=1178.359,192.713,-59.153,-177.927,6.759,148.639
C01430=1178.363,192.464,-59.130,-177.930,6.757,148.639
C01431=1178.368,192.215,-59.107,-177.932,6.755,148.639
C01432=1178.373,191.967,-59.083,-177.935,6.754,148.640
C01433=1178.377,191.718,-59.059,-177.938,6.751,148.640
C01434=1178.382,191.469,-59.036,-177.941,6.749,148.640
C01435=1178.386,191.220,-59.013,-177.943,6.747,148.641
C01436=1178.391,190.971,-58.990,-177.946,6.745,148.641
C01437=1178.395,190.722,-58.966,-177.949,6.744,148.641
C01438=1178.400,190.473,-58.942,-177.951,6.742,148.642
C01439=1178.404,190.224,-58.919,-177.954,6.739,148.642
C01440=1178.409,189.975,-58.896,-177.957,6.737,148.642
C01441=1178.414,189.726,-58.872,-177.959,6.735,148.643
C01442=1178.418,189.477,-58.849,-177.962,6.733,148.643
C01443=1178.423,189.229,-58.826,-177.965,6.732,148.643
C01444=1178.428,188.980,-58.803,-177.967,6.729,148.643
C01445=1178.432,188.731,-58.780,-177.970,6.727,148.644
C01446=1178.437,188.482,-58.756,-177.973,6.725,148.644
C01447=1178.442,188.233,-58.733,-177.975,6.723,148.644
C01448=1178.446,187.984,-58.710,-177.978,6.722,148.645
C01449=1178.451,187.735,-58.687,-177.981,6.720,148.645
C01450=1178.455,187.486,-58.664,-177.984,6.717,148.645
C01451=1178.460,187.237,-58.640,-177.986,6.715,148.646
C01452=1178.464,186.989,-58.618,-177.989,6.713,148.646
C01453=1178.469,186.740,-58.594,-177.992,6.712,148.646
C01454=1178.474,186.491,-58.571,-177.994,6.710,148.647
C01455=1178.479,186.242,-58.548,-177.997,6.708,148.647
C01456=1178.483,185.993,-58.525,-177.999,6.706,148.647
C01457=1178.487,185.744,-58.502,-178.002,6.703,148.647
C01458=1178.493,185.496,-58.479,-178.005,6.701,148.648
C01459=1178.497,185.247,-58.455,-178.008,6.700,148.648
C01460=1178.501,184.998,-58.433,-178.010,6.698,148.649
C01461=1178.507,184.729,-58.407,-178.013,6.696,148.649
C01462=1178.512,184.459,-58.382,-178.016,6.694,148.649
C01463=1178.516,184.189,-58.358,-178.019,6.692,148.650
C01464=1178.522,183.920,-58.333,-178.022,6.689,148.650
C01465=1178.526,183.671,-58.310,-178.025,6.687,148.650
C01466=1178.531,183.421,-58.288,-178.028,6.686,148.651
C01467=1178.535,183.172,-58.264,-178.030,6.683,148.651
C01468=1178.540,182.924,-58.242,-178.032,6.682,148.651
C01469=1178.545,182.675,-58.218,-178.035,6.680,148.651
C01470=1178.549,182.426,-58.195,-178.038,6.678,148.652
C01471=1178.554,182.177,-58.173,-178.041,6.676,148.652
C01472=1178.558,181.928,-58.150,-178.044,6.674,148.653
C01473=1178.563,181.680,-58.127,-178.046,6.672,148.653
C01474=1178.568,181.431,-58.104,-178.049,6.670,148.653
C01475=1178.573,181.181,-58.081,-178.051,6.668,148.653
C01476=1178.577,180.932,-58.058,-178.054,6.666,148.654
C01477=1178.582,180.684,-58.036,-178.057,6.665,148.654
C01478=1178.586,180.435,-58.013,-178.059,6.663,148.654
C01479=1178.591,180.186,-57.990,-178.063,6.660,148.655
C01480=1178.595,179.937,-57.967,-178.065,6.658,148.655
C01481=1178.600,179.688,-57.945,-178.068,6.657,148.656
C01482=1178.604,179.439,-57.922,-178.071,6.655,148.656
C01483=1178.609,179.190,-57.900,-178.073,6.653,148.656
C01484=1178.614,178.942,-57.877,-178.075,6.651,148.656
C01485=1178.619,178.692,-57.854,-178.078,6.649,148.657
C01486=1178.623,178.443,-57.832,-178.081,6.647,148.657
C01487=1178.628,178.194,-57.808,-178.083,6.646,148.657
C01488=1178.632,177.945,-57.787,-178.086,6.644,148.658
C01489=1178.637,177.696,-57.763,-178.089,6.641,148.658
C01490=1178.641,177.447,-57.741,-178.092,6.639,148.659
C01491=1178.647,177.199,-57.718,-178.095,6.638,148.659
C01492=1178.651,176.949,-57.696,-178.097,6.636,148.659
C01493=1178.656,176.700,-57.673,-178.100,6.634,148.659
C01494=1178.661,176.452,-57.651,-178.102,6.632,148.660
C01495=1178.665,176.203,-57.628,-178.105,6.630,148.660
C01496=1178.670,175.953,-57.606,-178.108,6.628,148.660
C01497=1178.674,175.705,-57.584,-178.110,6.627,148.661
C01498=1178.679,175.456,-57.561,-178.113,6.625,148.661
C01499=1178.683,175.207,-57.538,-178.116,6.623,148.662
C01500=1178.689,174.958,-57.516,-178.118,6.621,148.662
C01501=1178.693,174.709,-57.493,-178.121,6.620,148.662
C01502=1178.697,174.461,-57.471,-178.124,6.617,148.663
C01503=1178.703,174.211,-57.449,-178.127,6.615,148.663
C01504=1178.706,173.962,-57.426,-178.129,6.613,148.663
C01505=1178.711,173.714,-57.404,-178.132,6.611,148.664
C01506=1178.716,173.464,-57.382,-178.135,6.610,148.664
C01507=1178.720,173.215,-57.359,-178.137,6.608,148.664
C01508=1178.725,172.967,-57.337,-178.140,6.606,148.665
C01509=1178.730,172.717,-57.315,-178.143,6.604,148.665
C01510=1178.735,172.469,-57.292,-178.145,6.602,148.665
C01511=1178.739,172.220,-57.270,-178.148,6.601,148.666
C01512=1178.745,171.971,-57.248,-178.151,6.599,148.666
C01513=1178.749,171.722,-57.225,-178.153,6.597,148.666
C01514=1178.753,171.473,-57.203,-178.156,6.595,148.667
C01515=1178.758,171.224,-57.181,-178.159,6.594,148.667
C01516=1178.763,170.974,-57.159,-178.161,6.592,148.668
C01517=1178.767,170.726,-57.136,-178.164,6.590,148.668
C01518=1178.772,170.477,-57.114,-178.167,6.588,148.668
C01519=1178.777,170.228,-57.092,-178.169,6.587,148.669
C01520=1178.781,169.979,-57.070,-178.173,6.584,148.669
C01521=1178.786,169.730,-57.048,-178.175,6.582,148.669
C01522=1178.790,169.481,-57.025,-178.178,6.580,148.669
C01523=1178.796,169.232,-57.003,-178.180,6.578,148.670
C01524=1178.800,168.983,-56.981,-178.183,6.577,148.670
C01525=1178.805,168.734,-56.959,-178.186,6.575,148.671
C01526=1178.809,168.485,-56.937,-178.188,6.573,148.671
C01527=1178.814,168.236,-56.916,-178.191,6.571,148.671
C01528=1178.819,167.987,-56.893,-178.194,6.569,148.672
C01529=1178.824,167.738,-56.871,-178.196,6.568,148.672
C01530=1178.828,167.489,-56.849,-178.199,6.566,148.672
C01531=1178.833,167.241,-56.827,-178.202,6.564,148.673
C01532=1178.837,166.991,-56.805,-178.204,6.562,148.673
C01533=1178.842,166.743,-56.783,-178.207,6.561,148.674
C01534=1178.847,166.493,-56.761,-178.210,6.559,148.674
C01535=1178.852,166.244,-56.739,-178.212,6.557,148.674
C01536=1178.856,165.995,-56.717,-178.215,6.555,148.675
C01537=1178.861,165.747,-56.695,-178.218,6.554,148.675
C01538=1178.865,165.497,-56.673,-178.220,6.552,148.675
C01539=1178.870,165.249,-56.651,-178.223,6.550,148.676
C01540=1178.874,164.999,-56.629,-178.226,6.548,148.676
C01541=1178.879,164.751,-56.608,-178.228,6.546,148.676
C01542=1178.884,164.501,-56.586,-178.231,6.545,148.677
C01543=1178.888,164.253,-56.564,-178.234,6.543,148.677
C01544=1178.893,164.004,-56.542,-178.237,6.541,148.678
C01545=1178.898,163.754,-56.521,-178.239,6.539,148.678
C01546=1178.903,163.505,-56.499,-178.242,6.538,148.678
C01547=1178.908,163.256,-56.477,-178.245,6.536,148.679
C01548=1178.913,163.007,-56.455,-178.247,6.534,148.679
C01549=1178.917,162.758,-56.433,-178.250,6.532,148.679
C01550=1178.922,162.509,-56.411,-178.253,6.531,148.680
C01551=1178.927,162.260,-56.390,-178.255,6.529,148.680
C01552=1178.931,162.011,-56.367,-178.258,6.527,148.681
C01553=1178.936,161.762,-56.347,-178.261,6.525,148.681
C01554=1178.941,161.513,-56.325,-178.263,6.523,148.681
C01555=1178.945,161.264,-56.303,-178.266,6.522,148.682
C01556=1178.950,161.015,-56.281,-178.269,6.520,148.682
C01557=1178.954,160.766,-56.260,-178.271,6.518,148.682
C01558=1178.959,160.517,-56.239,-178.274,6.516,148.683
C01559=1178.964,160.268,-56.217,-178.277,6.515,148.683
C01560=1178.968,160.019,-56.195,-178.279,6.513,148.684
C01561=1178.973,159.770,-56.173,-178.282,6.511,148.684
C01562=1178.978,159.521,-56.152,-178.285,6.509,148.684
C01563=1178.982,159.272,-56.130,-178.288,6.508,148.685
C01564=1178.987,159.023,-56.109,-178.290,6.506,148.685
C01565=1178.993,158.754,-56.085,-178.293,6.504,148.686
C01566=1178.997,158.485,-56.062,-178.296,6.503,148.686
C01567=1179.002,158.216,-56.038,-178.299,6.501,148.686
C01568=1179.007,157.947,-56.016,-178.301,6.499,148.687
C01569=1179.012,157.698,-55.994,-178.304,6.497,148.687
C01570=1179.017,157.449,-55.973,-178.307,6.496,148.687
C01571=1179.022,157.200,-55.951,-178.310,6.494,148.688
C01572=1179.026,156.951,-55.931,-178.312,6.492,148.688
C01573=1179.031,156.702,-55.909,-178.315,6.490,148.689
C01574=1179.036,156.453,-55.887,-178.318,6.489,148.689
C01575=1179.040,156.203,-55.866,-178.321,6.487,148.690
C01576=1179.045,155.955,-55.844,-178.323,6.485,148.690
C01577=1179.050,155.705,-55.823,-178.326,6.484,148.690
C01578=1179.054,155.456,-55.802,-178.329,6.482,148.691
C01579=1179.059,155.207,-55.781,-178.332,6.480,148.691
C01580=1179.064,154.959,-55.759,-178.334,6.478,148.691
C01581=1179.069,154.710,-55.737,-178.337,6.477,148.692
C01582=1179.073,154.460,-55.716,-178.339,6.476,148.692
C01583=1179.077,154.212,-55.695,-178.342,6.474,148.693
C01584=1179.083,153.962,-55.674,-178.344,6.472,148.693
C01585=1179.088,153.713,-55.653,-178.347,6.470,148.693
C01586=1179.092,153.464,-55.631,-178.350,6.469,148.694
C01587=1179.097,153.215,-55.611,-178.352,6.467,148.694
C01588=1179.101,152.966,-55.589,-178.355,6.465,148.694
C01589=1179.107,152.717,-55.568,-178.358,6.463,148.695
C01590=1179.111,152.468,-55.546,-178.361,6.462,148.695
C01591=1179.115,152.219,-55.526,-178.364,6.460,148.696
C01592=1179.120,151.970,-55.504,-178.366,6.458,148.696
C01593=1179.125,151.721,-55.483,-178.369,6.457,148.697
C01594=1179.130,151.472,-55.463,-178.372,6.455,148.697
C01595=1179.135,151.223,-55.441,-178.374,6.454,148.697
C01596=1179.140,150.974,-55.420,-178.377,6.452,148.698
C01597=1179.144,150.724,-55.399,-178.379,6.450,148.698
C01598=1179.149,150.476,-55.377,-178.382,6.449,148.699
C01599=1179.154,150.226,-55.357,-178.385,6.447,148.699
C01600=1179.158,149.977,-55.336,-178.387,6.445,148.699
C01601=1179.163,149.729,-55.314,-178.390,6.443,148.700
C01602=1179.168,149.479,-55.294,-178.393,6.442,148.700
C01603=1179.172,149.230,-55.273,-178.396,6.440,148.701
C01604=1179.177,148.981,-55.252,-178.399,6.438,148.701
C01605=1179.182,148.732,-55.230,-178.401,6.437,148.701
C01606=1179.186,148.483,-55.210,-178.403,6.436,148.702
C01607=1179.192,148.234,-55.189,-178.406,6.434,148.702
C01608=1179.196,147.985,-55.168,-178.409,6.432,148.703
C01609=1179.201,147.736,-55.147,-178.411,6.430,148.703
C01610=1179.205,147.486,-55.126,-178.414,6.429,148.703
C01611=1179.210,147.237,-55.105,-178.417,6.427,148.704
C01612=1179.215,146.988,-55.084,-178.420,6.426,148.704
C01613=1179.220,146.739,-55.064,-178.422,6.425,148.705
C01614=1179.224,146.490,-55.042,-178.425,6.423,148.705
C01615=1179.229,146.241,-55.022,-178.427,6.421,148.705
C01616=1179.234,145.992,-55.001,-178.430,6.419,148.706
C01617=1179.239,145.743,-54.980,-178.433,6.418,148.706
C01618=1179.244,145.494,-54.959,-178.436,6.416,148.707
C01619=1179.248,145.245,-54.939,-178.438,6.414,148.707
C01620=1179.253,144.996,-54.918,-178.441,6.413,148.708
C01621=1179.258,144.747,-54.898,-178.444,6.412,148.708
C01622=1179.262,144.497,-54.876,-178.446,6.410,148.708
C01623=1179.266,144.249,-54.855,-178.449,6.408,148.709
C01624=1179.272,143.999,-54.834,-178.452,6.406,148.709
C01625=1179.276,143.750,-54.814,-178.454,6.405,148.710
C01626=1179.281,143.501,-54.793,-178.457,6.403,148.710
C01627=1179.286,143.252,-54.773,-178.460,6.402,148.711
C01628=1179.290,143.003,-54.752,-178.462,6.401,148.711
C01629=1179.295,142.754,-54.731,-178.465,6.399,148.711
C01630=1179.300,142.505,-54.711,-178.468,6.397,148.712
C01631=1179.305,142.256,-54.690,-178.470,6.395,148.712
C01632=1179.309,142.007,-54.669,-178.473,6.394,148.712
C01633=1179.315,141.757,-54.648,-178.476,6.392,148.713
C01634=1179.319,141.509,-54.628,-178.478,6.391,148.713
C01635=1179.323,141.260,-54.608,-178.481,6.389,148.714
C01636=1179.329,141.010,-54.587,-178.484,6.388,148.714
C01637=1179.333,140.761,-54.567,-178.486,6.386,148.715
C01638=1179.338,140.512,-54.547,-178.489,6.384,148.715
C01639=1179.343,140.263,-54.526,-178.492,6.382,148.715
C01640=1179.347,140.014,-54.505,-178.495,6.381,148.716
C01641=1179.353,139.764,-54.484,-178.497,6.380,148.716
C01642=1179.357,139.515,-54.464,-178.500,6.378,148.717
C01643=1179.361,139.266,-54.444,-178.503,6.377,148.717
C01644=1179.367,139.017,-54.423,-178.505,6.375,148.718
C01645=1179.371,138.768,-54.403,-178.508,6.373,148.718
C01646=1179.376,138.519,-54.383,-178.510,6.372,148.718
C01647=1179.380,138.270,-54.362,-178.513,6.371,148.719
C01648=1179.385,138.020,-54.341,-178.516,6.369,148.719
C01649=1179.390,137.771,-54.321,-178.519,6.367,148.720
C01650=1179.395,137.523,-54.302,-178.521,6.366,148.720
C01651=1179.400,137.273,-54.281,-178.524,6.364,148.721
C01652=1179.405,137.024,-54.260,-178.526,6.363,148.721
C01653=1179.409,136.775,-54.240,-178.529,6.361,148.722
C01654=1179.414,136.526,-54.220,-178.532,6.360,148.722
C01655=1179.419,136.277,-54.199,-178.535,6.358,148.722
C01656=1179.424,136.028,-54.179,-178.537,6.356,148.723
C01657=1179.428,135.779,-54.159,-178.540,6.355,148.723
C01658=1179.433,135.529,-54.139,-178.543,6.354,148.724
C01659=1179.438,135.280,-54.118,-178.545,6.352,148.724
C01660=1179.442,135.031,-54.098,-178.548,6.350,148.724
C01661=1179.448,134.782,-54.078,-178.551,6.349,148.725
C01662=1179.452,134.533,-54.058,-178.553,6.348,148.725
C01663=1179.457,134.284,-54.038,-178.556,6.346,148.726
C01664=1179.462,134.034,-54.017,-178.559,6.345,148.726
C01665=1179.466,133.785,-53.997,-178.561,6.343,148.727
C01666=1179.471,133.536,-53.977,-178.564,6.341,148.727
C01667=1179.476,133.287,-53.957,-178.566,6.340,148.727
C01668=1179.481,133.039,-53.937,-178.569,6.339,148.728
C01669=1179.486,132.770,-53.915,-178.572,6.337,148.728
C01670=1179.491,132.501,-53.894,-178.575,6.335,148.729
C01671=1179.496,132.232,-53.871,-178.578,6.334,148.729
C01672=1179.501,131.963,-53.850,-178.581,6.332,148.730
C01673=1179.506,131.715,-53.830,-178.583,6.330,148.730
C01674=1179.511,131.465,-53.811,-178.586,6.329,148.731
C01675=1179.515,131.217,-53.790,-178.589,6.328,148.731
C01676=1179.521,130.967,-53.770,-178.591,6.326,148.732
C01677=1179.525,130.718,-53.750,-178.594,6.325,148.732
C01678=1179.530,130.469,-53.730,-178.597,6.323,148.732
C01679=1179.535,130.220,-53.710,-178.599,6.322,148.733
C01680=1179.540,129.970,-53.690,-178.602,6.320,148.733
C01681=1179.544,129.721,-53.670,-178.605,6.319,148.734
C01682=1179.549,129.472,-53.650,-178.608,6.317,148.734
C01683=1179.554,129.223,-53.631,-178.610,6.316,148.735
C01684=1179.559,128.974,-53.611,-178.613,6.315,148.735
C01685=1179.563,128.724,-53.591,-178.616,6.313,148.736
C01686=1179.568,128.475,-53.571,-178.618,6.311,148.736
C01687=1179.573,128.227,-53.551,-178.621,6.309,148.736
C01688=1179.578,127.977,-53.532,-178.624,6.309,148.737
C01689=1179.582,127.728,-53.511,-178.626,6.307,148.737
C01690=1179.587,127.479,-53.492,-178.629,6.305,148.738
C01691=1179.592,127.230,-53.472,-178.631,6.304,148.738
C01692=1179.597,126.981,-53.452,-178.634,6.303,148.739
C01693=1179.602,126.731,-53.432,-178.637,6.301,148.739
C01694=1179.606,126.482,-53.413,-178.640,6.300,148.740
C01695=1179.611,126.233,-53.393,-178.642,6.299,148.740
C01696=1179.616,125.984,-53.373,-178.645,6.297,148.741
C01697=1179.621,125.734,-53.353,-178.648,6.296,148.741
C01698=1179.626,125.486,-53.333,-178.650,6.294,148.742
C01699=1179.631,125.236,-53.314,-178.653,6.293,148.742
C01700=1179.635,124.987,-53.294,-178.656,6.291,148.743
C01701=1179.640,124.737,-53.274,-178.658,6.290,148.743
C01702=1179.644,124.489,-53.255,-178.661,6.288,148.743
C01703=1179.649,124.240,-53.235,-178.663,6.287,148.744
C01704=1179.654,123.990,-53.216,-178.666,6.286,148.744
C01705=1179.659,123.741,-53.196,-178.669,6.284,148.745
C01706=1179.664,123.492,-53.177,-178.671,6.283,148.745
C01707=1179.668,123.243,-53.156,-178.674,6.281,148.746
C01708=1179.674,122.994,-53.137,-178.677,6.280,148.746
C01709=1179.678,122.744,-53.117,-178.680,6.278,148.747
C01710=1179.682,122.495,-53.098,-178.682,6.277,148.747
C01711=1179.688,122.246,-53.079,-178.685,6.275,148.747
C01712=1179.693,121.997,-53.059,-178.688,6.274,148.748
C01713=1179.697,121.747,-53.040,-178.690,6.273,148.748
C01714=1179.702,121.499,-53.020,-178.693,6.271,148.749
C01715=1179.707,121.249,-53.000,-178.695,6.270,148.749
C01716=1179.711,121.000,-52.981,-178.699,6.268,148.750
C01717=1179.716,120.751,-52.962,-178.701,6.267,148.750
C01718=1179.721,120.502,-52.942,-178.703,6.266,148.751
C01719=1179.726,120.253,-52.923,-178.707,6.264,148.751
C01720=1179.731,120.003,-52.903,-178.709,6.263,148.752
C01721=1179.735,119.754,-52.884,-178.711,6.262,148.752
C01722=1179.741,119.505,-52.865,-178.714,6.260,148.752
C01723=1179.745,119.255,-52.845,-178.717,6.259,148.753
C01724=1179.751,119.007,-52.826,-178.719,6.258,148.754
C01725=1179.755,118.757,-52.807,-178.722,6.256,148.754
C01726=1179.759,118.508,-52.787,-178.725,6.255,148.755
C01727=1179.765,118.259,-52.768,-178.727,6.254,148.755
C01728=1179.770,118.009,-52.748,-178.730,6.252,148.755
C01729=1179.774,117.761,-52.729,-178.733,6.250,148.756
C01730=1179.779,117.511,-52.710,-178.735,6.249,148.756
C01731=1179.784,117.262,-52.691,-178.738,6.248,148.757
C01732=1179.788,117.013,-52.671,-178.741,6.246,148.757
C01733=1179.793,116.764,-52.652,-178.744,6.245,148.758
C01734=1179.798,116.515,-52.633,-178.746,6.244,148.758
C01735=1179.803,116.265,-52.613,-178.749,6.242,148.759
C01736=1179.808,116.016,-52.595,-178.752,6.241,148.759
C01737=1179.813,115.766,-52.575,-178.754,6.240,148.760
C01738=1179.818,115.517,-52.556,-178.757,6.238,148.760
C01739=1179.822,115.268,-52.537,-178.759,6.237,148.760
C01740=1179.827,115.019,-52.518,-178.762,6.236,148.761
C01741=1179.831,114.770,-52.499,-178.765,6.234,148.761
C01742=1179.837,114.521,-52.480,-178.767,6.233,148.762
C01743=1179.842,114.271,-52.460,-178.770,6.232,148.763
C01744=1179.846,114.022,-52.442,-178.773,6.230,148.763
C01745=1179.851,113.773,-52.422,-178.775,6.229,148.763
C01746=1179.856,113.524,-52.403,-178.778,6.228,148.764
C01747=1179.861,113.274,-52.384,-178.780,6.227,148.764
C01748=1179.866,113.025,-52.365,-178.783,6.225,148.765
C01749=1179.870,112.776,-52.346,-178.786,6.224,148.765
C01750=1179.875,112.527,-52.327,-178.788,6.223,148.766
C01751=1179.880,112.277,-52.308,-178.791,6.221,148.766
C01752=1179.885,112.028,-52.289,-178.794,6.219,148.767
C01753=1179.890,111.779,-52.269,-178.797,6.219,148.767
C01754=1179.894,111.530,-52.251,-178.799,6.217,148.768
C01755=1179.900,111.281,-52.232,-178.802,6.215,148.768
C01756=1179.904,111.032,-52.213,-178.805,6.215,148.769
C01757=1179.909,110.783,-52.194,-178.807,6.213,148.769
C01758=1179.914,110.533,-52.175,-178.810,6.211,148.770
C01759=1179.919,110.284,-52.156,-178.813,6.211,148.770
C01760=1179.923,110.035,-52.137,-178.815,6.209,148.771
C01761=1179.929,109.785,-52.118,-178.818,6.208,148.771
C01762=1179.933,109.536,-52.099,-178.821,6.206,148.772
C01763=1179.938,109.286,-52.081,-178.823,6.205,148.772
C01764=1179.943,109.038,-52.062,-178.826,6.204,148.773
C01765=1179.948,108.788,-52.042,-178.829,6.202,148.773
C01766=1179.953,108.539,-52.025,-178.831,6.201,148.773
C01767=1179.957,108.290,-52.005,-178.834,6.200,148.774
C01768=1179.962,108.040,-51.987,-178.837,6.198,148.775
C01769=1179.967,107.792,-51.968,-178.839,6.198,148.775
C01770=1179.972,107.542,-51.949,-178.842,6.196,148.776
C01771=1179.977,107.293,-51.931,-178.845,6.194,148.776
C01772=1179.982,107.043,-51.912,-178.847,6.194,148.776
C01773=1179.986,106.775,-51.891,-178.850,6.192,148.777
C01774=1179.992,106.507,-51.871,-178.853,6.190,148.777
C01775=1179.998,106.239,-51.851,-178.856,6.189,148.778
C01776=1180.002,105.970,-51.831,-178.858,6.188,148.778
C01777=1180.007,105.721,-51.813,-178.861,6.187,148.779
C01778=1180.013,105.472,-51.794,-178.864,6.185,148.780
C01779=1180.017,105.222,-51.775,-178.867,6.184,148.780
C01780=1180.022,104.973,-51.756,-178.869,6.183,148.781
C01781=1180.027,104.724,-51.738,-178.871,6.182,148.781
C01782=1180.031,104.475,-51.719,-178.875,6.180,148.782
C01783=1180.037,104.225,-51.700,-178.877,6.179,148.782
C01784=1180.042,103.976,-51.682,-178.879,6.178,148.782
C01785=1180.046,103.727,-51.663,-178.883,6.176,148.783
C01786=1180.051,103.477,-51.645,-178.885,6.176,148.784
C01787=1180.056,103.229,-51.626,-178.888,6.174,148.784
C01788=1180.060,102.979,-51.608,-178.891,6.172,148.785
C01789=1180.066,102.729,-51.589,-178.893,6.172,148.785
C01790=1180.070,102.481,-51.571,-178.896,6.170,148.786
C01791=1180.075,102.231,-51.552,-178.898,6.169,148.786
C01792=1180.080,101.982,-51.534,-178.901,6.168,148.786
C01793=1180.085,101.733,-51.515,-178.903,6.167,148.787
C01794=1180.090,101.484,-51.497,-178.906,6.165,148.787
C01795=1180.094,101.234,-51.479,-178.909,6.164,148.788
C01796=1180.099,100.985,-51.461,-178.912,6.163,148.789
C01797=1180.105,100.736,-51.441,-178.914,6.161,148.789
C01798=1180.109,100.486,-51.423,-178.917,6.161,148.790
C01799=1180.114,100.237,-51.405,-178.920,6.159,148.790
C01800=1180.119,99.987,-51.387,-178.922,6.158,148.790
C01801=1180.124,99.739,-51.368,-178.925,6.157,148.791
C01802=1180.128,99.489,-51.349,-178.928,6.155,148.791
C01803=1180.133,99.240,-51.331,-178.930,6.154,148.792
C01804=1180.138,98.990,-51.313,-178.933,6.153,148.793
C01805=1180.143,98.741,-51.295,-178.935,6.152,148.793
C01806=1180.148,98.492,-51.276,-178.938,6.150,148.794
C01807=1180.153,98.242,-51.258,-178.940,6.150,148.794
C01808=1180.158,97.993,-51.240,-178.944,6.148,148.795
C01809=1180.163,97.744,-51.222,-178.946,6.147,148.795
